Yaskawa INFORM job: DPRINT3D8.JBI

/JOB
//NAME DPRINT3D8
//POS
///NPOS 990,0,0,0,0,0
///TOOL 9
///POSTYPE PULSE
///PULSE
C00000=29490,52359,-120568,61658,-120234,-93746,0
C00001=29537,52361,-120565,61607,-120252,-93751,0
C00002=29592,52361,-120565,61546,-120272,-93759,0
C00003=29651,52358,-120574,61480,-120290,-93771,0
C00004=29730,52355,-120589,61392,-120313,-93786,0
C00005=29809,52348,-120612,61302,-120332,-93804,0
C00006=29942,52328,-120680,61146,-120353,-93842,0
C00007=30018,52314,-120729,61056,-120361,-93866,0
C00008=30112,52288,-120820,60939,-120358,-93905,0
C00009=30203,52259,-120919,60825,-120351,-93946,0
C00010=30285,52224,-121037,60719,-120333,-93990,0
C00011=30363,52187,-121164,60616,-120310,-94037,0
C00012=30429,52145,-121304,60523,-120276,-94086,0
C00013=30490,52102,-121452,60436,-120237,-94135,0
C00014=30538,52055,-121611,60361,-120190,-94186,0
C00015=30572,52018,-121739,60306,-120149,-94227,0
C00016=30580,52008,-121774,60292,-120138,-94237,0
C00017=30594,51982,-121860,60265,-120107,-94263,0
C00018=30605,51957,-121946,60241,-120076,-94288,0
C00019=30621,51904,-122127,60198,-120009,-94341,0
C00020=30624,51867,-122253,60178,-119957,-94376,0
C00021=30621,51830,-122380,60164,-119904,-94411,0
C00022=30618,51802,-122475,60155,-119864,-94437,0
C00023=30609,51776,-122563,60152,-119825,-94460,0
C00024=30600,51755,-122637,60152,-119791,-94479,0
C00025=30571,51703,-122814,60160,-119709,-94524,0
C00026=30542,51669,-122932,60176,-119650,-94553,0
C00027=30510,51638,-123039,60197,-119595,-94579,0
C00028=30482,51612,-123127,60216,-119549,-94600,0
C00029=30451,51588,-123208,60240,-119505,-94618,0
C00030=30396,51554,-123325,60285,-119439,-94643,0
C00031=30357,51531,-123404,60318,-119393,-94659,0
C00032=30314,51511,-123476,60355,-119349,-94673,0
C00033=30248,51483,-123570,60415,-119289,-94691,0
C00034=30201,51465,-123633,60459,-119247,-94702,0
C00035=30148,51448,-123692,60510,-119205,-94711,0
C00036=30074,51428,-123761,60583,-119152,-94720,0
C00037=30016,51413,-123811,60640,-119112,-94727,0
C00038=29954,51400,-123854,60703,-119074,-94730,0
C00039=29879,51388,-123894,60780,-119033,-94731,0
C00040=29815,51379,-123926,60847,-118999,-94732,0
C00041=29746,51372,-123949,60920,-118966,-94730,0
C00042=29673,51367,-123964,60998,-118936,-94724,0
C00043=29603,51364,-123975,61074,-118908,-94718,0
C00044=29535,51363,-123978,61148,-118885,-94709,0
C00045=29463,51364,-123971,61228,-118864,-94698,0
C00046=29411,51366,-123964,61286,-118849,-94689,0
C00047=29309,51372,-123940,61403,-118825,-94669,0
C00048=29207,51381,-123905,61519,-118804,-94646,0
C00049=29109,51397,-123850,61634,-118794,-94617,0
C00050=29015,51415,-123785,61747,-118788,-94586,0
C00051=28926,51438,-123701,61855,-118793,-94550,0
C00052=28842,51464,-123609,61960,-118801,-94513,0
C00053=28766,51495,-123499,62057,-118819,-94471,0
C00054=28695,51529,-123383,62150,-118841,-94429,0
C00055=28635,51566,-123252,62233,-118872,-94384,0
C00056=28581,51605,-123115,62311,-118908,-94338,0
C00057=28539,51647,-122969,62376,-118951,-94291,0
C00058=28503,51691,-122818,62435,-118997,-94243,0
C00059=28481,51736,-122661,62481,-119051,-94195,0
C00060=28464,51782,-122502,62520,-119109,-94148,0
C00061=28461,51829,-122341,62545,-119170,-94102,0
C00062=28463,51859,-122240,62556,-119210,-94073,0
C00063=28476,51924,-122018,62572,-119302,-94012,0
C00064=28493,51964,-121883,62572,-119360,-93976,0
C00065=28528,52017,-121701,62558,-119443,-93930,0
C00066=28561,52056,-121571,62539,-119506,-93897,0
C00067=28618,52106,-121405,62499,-119591,-93858,0
C00068=28668,52142,-121282,62461,-119657,-93830,0
C00069=28743,52185,-121137,62399,-119740,-93800,0
C00070=28808,52218,-121030,62342,-119805,-93779,0
C00071=28898,52253,-120912,62259,-119885,-93758,0
C00072=28977,52280,-120825,62185,-119948,-93744,0
C00073=29075,52306,-120741,62090,-120016,-93735,0
C00074=29171,52330,-120661,61995,-120081,-93726,0
C00075=25221,55476,-110646,67744,-122004,-90321,0
C00076=36362,52521,-120169,76431,-115202,-92037,0
C00077=36363,52459,-120191,76439,-115220,-92015,0
C00078=23322,59783,-98074,71828,-124780,-86450,0
C00079=23300,59778,-98087,71848,-124763,-86450,0
C00080=23207,59762,-98132,71934,-124696,-86448,0
C00081=23134,59755,-98149,72005,-124649,-86441,0
C00082=23037,59755,-98149,72103,-124591,-86425,0
C00083=22967,59761,-98132,72177,-124555,-86408,0
C00084=22871,59777,-98086,72281,-124511,-86380,0
C00085=22816,59791,-98047,72343,-124489,-86360,0
C00086=22729,59817,-97973,72444,-124458,-86325,0
C00087=22655,59848,-97887,72533,-124437,-86289,0
C00088=22584,59883,-97789,72621,-124421,-86250,0
C00089=22520,59926,-97670,72707,-124416,-86206,0
C00090=22458,59972,-97541,72791,-124413,-86159,0
C00091=22405,60025,-97394,72870,-124420,-86109,0
C00092=22356,60081,-97239,72947,-124432,-86057,0
C00093=22316,60142,-97070,73016,-124452,-86003,0
C00094=22280,60206,-96894,73082,-124478,-85948,0
C00095=22255,60273,-96709,73140,-124512,-85891,0
C00096=22235,60342,-96520,73194,-124549,-85835,0
C00097=22226,60412,-96326,73237,-124595,-85779,0
C00098=22221,60483,-96130,73276,-124643,-85722,0
C00099=22228,60555,-95934,73304,-124698,-85668,0
C00100=22235,60601,-95807,73320,-124736,-85633,0
C00101=22239,60626,-95740,73327,-124756,-85615,0
C00102=22260,60696,-95549,73341,-124818,-85565,0
C00103=22280,60753,-95392,73349,-124872,-85524,0
C00104=22317,60832,-95177,73351,-124950,-85469,0
C00105=22350,60886,-95029,73345,-125009,-85433,0
C00106=22403,60957,-94836,73326,-125091,-85387,0
C00107=22449,61008,-94699,73306,-125156,-85357,0
C00108=22516,61067,-94539,73269,-125238,-85322,0
C00109=22573,61109,-94424,73234,-125304,-85299,0
C00110=22650,61156,-94298,73180,-125384,-85277,0
C00111=22717,61189,-94210,73130,-125449,-85263,0
C00112=22802,61220,-94125,73061,-125523,-85253,0
C00113=22876,61242,-94068,72999,-125584,-85250,0
C00114=22965,61257,-94026,72917,-125651,-85253,0
C00115=22998,61262,-94015,72887,-125674,-85256,0
C00116=23044,61265,-94005,72844,-125705,-85261,0
C00117=23092,61265,-94006,72795,-125735,-85269,0
C00118=23153,61264,-94010,72735,-125772,-85281,0
C00119=23215,61259,-94025,72670,-125806,-85295,0
C00120=23304,61242,-94071,72574,-125849,-85324,0
C00121=23341,61233,-94096,72532,-125866,-85336,0
C00122=23382,61222,-94128,72485,-125882,-85353,0
C00123=23426,61205,-94174,72433,-125897,-85373,0
C00124=23485,61181,-94239,72362,-125916,-85401,0
C00125=23541,61155,-94311,72293,-125931,-85431,0
C00126=23615,61108,-94439,72195,-125943,-85480,0
C00127=23682,61057,-94580,72103,-125945,-85531,0
C00128=23740,60998,-94741,72014,-125938,-85586,0
C00129=23795,60936,-94911,71928,-125926,-85643,0
C00130=23805,60920,-94953,71910,-125920,-85657,0
C00131=23839,60868,-95097,71849,-125901,-85702,0
C00132=23879,60798,-95289,71773,-125874,-85763,0
C00133=23909,60724,-95491,71706,-125836,-85825,0
C00134=23933,60649,-95698,71644,-125795,-85887,0
C00135=23946,60571,-95910,71592,-125744,-85949,0
C00136=23947,60554,-95958,71582,-125731,-85962,0
C00137=23949,60494,-96123,71549,-125688,-86009,0
C00138=23946,60453,-96234,71532,-125656,-86040,0
C00139=23942,60416,-96335,71518,-125625,-86067,0
C00140=23926,60337,-96554,71493,-125556,-86125,0
C00141=23909,60283,-96701,71484,-125504,-86164,0
C00142=23887,60231,-96843,71480,-125452,-86200,0
C00143=23870,60192,-96951,71478,-125412,-86227,0
C00144=23849,60157,-97049,71481,-125373,-86251,0
C00145=23831,60129,-97125,71485,-125342,-86269,0
C00146=23781,60061,-97311,71501,-125260,-86313,0
C00147=23731,60007,-97459,71526,-125189,-86346,0
C00148=23666,59949,-97619,71563,-125107,-86380,0
C00149=23605,59906,-97737,71603,-125038,-86403,0
C00150=23529,59861,-97861,71657,-124959,-86425,0
C00151=23459,59829,-97949,71712,-124895,-86438,0
C00152=23402,59808,-98007,71760,-124844,-86445,0
C00153=23317,59765,-98126,71824,-124763,-86464,0
C00154=35332,54396,-113967,78226,-116318,-89994,0
C00155=36295,54803,-112729,77380,-117083,-89721,0
C00156=40947,51674,-122953,71228,-116241,-93341,0
C00157=33828,55772,-109747,58612,-126255,-91536,0
C00158=35387,54350,-114111,78152,-116309,-90043,0
C00159=35603,55084,-111856,78200,-116951,-89383,0
C00160=36476,55477,-110686,77450,-117670,-89127,0
C00161=42174,51641,-123098,69885,-116652,-93519,0
C00162=33600,55094,-111787,58512,-125351,-92026,0
C00163=34232,54514,-113579,79405,-115874,-89764,0
C00164=35133,54883,-112462,78609,-116575,-89515,0
C00165=34898,55093,-111816,78927,-116607,-89295,0
C00166=35366,55295,-111211,78521,-116983,-89162,0
C00167=35549,55132,-111710,78273,-116958,-89333,0
C00168=36108,54854,-112568,77592,-117031,-89652,0
C00169=34832,55352,-111030,57280,-126168,-92063,0
C00170=36949,53594,-116517,54010,-124665,-93861,0
C00171=39301,53631,-116452,73778,-117508,-91183,0
C00172=44249,56266,-108496,69707,-122168,-89514,0
C00173=34852,55334,-111085,79062,-116751,-89069,0
C00174=32937,57301,-105238,81692,-116962,-87111,0
C00175=36072,54385,-114015,77455,-116661,-90086,0
C00176=40136,51651,-123013,72093,-115916,-93273,0
C00177=48633,53267,-117848,63578,-120957,-92820,0
C00178=48723,53302,-117737,63496,-121033,-92802,0
C00179=48757,53314,-117700,63465,-121059,-92797,0
C00180=48805,53330,-117652,63419,-121097,-92790,0
C00181=48859,53343,-117610,63367,-121134,-92786,0
C00182=48926,53359,-117560,63301,-121178,-92782,0
C00183=48998,53374,-117515,63229,-121223,-92781,0
C00184=49105,53388,-117471,63119,-121282,-92785,0
C00185=49151,53393,-117456,63070,-121305,-92788,0
C00186=49204,53398,-117444,63015,-121330,-92792,0
C00187=49261,53399,-117440,62953,-121354,-92800,0
C00188=49339,53401,-117437,62868,-121386,-92810,0
C00189=49415,53400,-117441,62784,-121414,-92824,0
C00190=49524,53391,-117472,62661,-121444,-92848,0
C00191=49626,53378,-117520,62542,-121467,-92877,0
C00192=49724,53357,-117590,62425,-121478,-92911,0
C00193=49819,53332,-117670,62309,-121484,-92948,0
C00194=49839,53326,-117692,62283,-121484,-92958,0
C00195=49907,53302,-117771,62197,-121480,-92989,0
C00196=49992,53269,-117880,62088,-121470,-93032,0
C00197=50067,53230,-118008,61987,-121451,-93079,0
C00198=50138,53189,-118144,61889,-121426,-93128,0
C00199=50198,53143,-118293,61802,-121390,-93178,0
C00200=50209,53132,-118329,61784,-121381,-93190,0
C00201=50247,53094,-118453,61723,-121347,-93230,0
C00202=50268,53068,-118539,61688,-121322,-93257,0
C00203=50285,53043,-118620,61657,-121297,-93282,0
C00204=50316,52988,-118800,61597,-121238,-93336,0
C00205=50330,52950,-118927,61564,-121193,-93374,0
C00206=50337,52911,-119054,61536,-121147,-93410,0
C00207=50342,52881,-119151,61517,-121111,-93438,0
C00208=50342,52853,-119244,61504,-121074,-93464,0
C00209=50339,52830,-119318,61496,-121045,-93483,0
C00210=50326,52774,-119503,61483,-120967,-93533,0
C00211=50304,52726,-119660,61485,-120897,-93573,0
C00212=50269,52672,-119839,61498,-120814,-93617,0
C00213=50230,52628,-119982,61521,-120744,-93652,0
C00214=50175,52579,-120143,61558,-120660,-93688,0
C00215=50119,52540,-120271,61602,-120590,-93715,0
C00216=50043,52496,-120413,61664,-120507,-93744,0
C00217=49976,52465,-120515,61724,-120443,-93763,0
C00218=49884,52430,-120630,61809,-120364,-93782,0
C00219=49808,52406,-120707,61882,-120306,-93793,0
C00220=49702,52380,-120791,61986,-120236,-93801,0
C00221=49621,52365,-120839,62069,-120188,-93803,0
C00222=49505,52350,-120888,62189,-120127,-93800,0
C00223=49436,52344,-120906,62262,-120095,-93795,0
C00224=49322,52337,-120926,62384,-120047,-93785,0
C00225=49222,52336,-120924,62495,-120011,-93770,0
C00226=49121,52339,-120912,62607,-119980,-93753,0
C00227=49023,52349,-120879,62720,-119957,-93729,0
C00228=48926,52361,-120834,62832,-119939,-93703,0
C00229=48834,52380,-120769,62942,-119930,-93672,0
C00230=48744,52401,-120695,63050,-119926,-93638,0
C00231=48662,52428,-120602,63154,-119932,-93600,0
C00232=48584,52458,-120499,63253,-119942,-93560,0
C00233=48514,52493,-120382,63346,-119961,-93518,0
C00234=48450,52530,-120257,63433,-119984,-93473,0
C00235=48397,52571,-120118,63511,-120017,-93426,0
C00236=48349,52614,-119974,63583,-120053,-93379,0
C00237=48314,52660,-119821,63644,-120097,-93331,0
C00238=48294,52691,-119719,63680,-120128,-93299,0
C00239=48284,52708,-119665,63698,-120145,-93282,0
C00240=48265,52756,-119504,63741,-120198,-93234,0
C00241=48254,52798,-119367,63773,-120245,-93194,0
C00242=48249,52857,-119173,63806,-120315,-93138,0
C00243=48254,52900,-119033,63821,-120369,-93099,0
C00244=48272,52958,-118841,63828,-120448,-93048,0
C00245=48294,53002,-118699,63825,-120508,-93010,0
C00246=48334,53058,-118519,63807,-120591,-92965,0
C00247=48372,53100,-118383,63785,-120657,-92932,0
C00248=48432,53151,-118221,63743,-120739,-92895,0
C00249=48487,53190,-118095,63702,-120807,-92868,0
C00250=48559,53231,-117963,63642,-120884,-92842,0
C00251=48631,53272,-117834,63582,-120961,-92816,0
C00252=30446,52027,-121515,60488,-120235,-94120,0
C00253=30497,51984,-121663,60411,-120192,-94169,0
C00254=30538,51942,-121805,60346,-120149,-94214,0
C00255=30574,51891,-121979,60283,-120090,-94267,0
C00256=30585,51872,-122044,60262,-120068,-94286,0
C00257=30597,51845,-122135,60236,-120035,-94314,0
C00258=30605,51817,-122231,60215,-119998,-94341,0
C00259=30612,51782,-122353,60190,-119951,-94376,0
C00260=30615,51745,-122479,60170,-119899,-94412,0
C00261=30606,51692,-122661,60155,-119822,-94460,0
C00262=30599,51669,-122738,60152,-119788,-94481,0
C00263=30589,51644,-122824,60152,-119749,-94503,0
C00264=30572,51617,-122915,60158,-119706,-94527,0
C00265=30548,51581,-123038,60168,-119648,-94557,0
C00266=30520,51547,-123156,60184,-119589,-94586,0
C00267=30465,51501,-123316,60223,-119504,-94624,0
C00268=30402,51458,-123462,60273,-119424,-94655,0
C00269=30327,51420,-123592,60338,-119344,-94682,0
C00270=30246,51384,-123715,60411,-119267,-94705,0
C00271=30226,51377,-123740,60430,-119250,-94709,0
C00272=30156,51354,-123820,60497,-119194,-94722,0
C00273=30061,51326,-123916,60589,-119124,-94735,0
C00274=29958,51304,-123990,60692,-119058,-94743,0
C00275=29853,51285,-124056,60800,-118997,-94747,0
C00276=29742,51272,-124098,60916,-118943,-94744,0
C00277=29718,51270,-124104,60943,-118932,-94742,0
C00278=29630,51265,-124121,61037,-118896,-94736,0
C00279=29571,51263,-124125,61102,-118876,-94729,0
C00280=29517,51264,-124124,61162,-118858,-94722,0
C00281=29399,51267,-124111,61293,-118824,-94702,0
C00282=29319,51273,-124088,61385,-118807,-94685,0
C00283=29241,51281,-124057,61475,-118793,-94666,0
C00284=29181,51288,-124031,61544,-118784,-94651,0
C00285=29126,51297,-123998,61608,-118778,-94634,0
C00286=29084,51305,-123970,61659,-118776,-94621,0
C00287=28979,51329,-123886,61785,-118774,-94583,0
C00288=28894,51353,-123799,61889,-118780,-94547,0
C00289=28802,51385,-123685,62006,-118795,-94502,0
C00290=28732,51416,-123574,62097,-118815,-94462,0
C00291=28656,51457,-123434,62199,-118845,-94412,0
C00292=28603,51493,-123308,62273,-118877,-94369,0
C00293=28547,51540,-123145,62357,-118922,-94315,0
C00294=28512,51579,-123009,62413,-118963,-94272,0
C00295=28478,51630,-122831,62474,-119021,-94217,0
C00296=28461,51671,-122690,62511,-119071,-94174,0
C00297=28450,51726,-122502,62548,-119140,-94119,0
C00298=28451,51766,-122363,62565,-119195,-94080,0
C00299=28464,51822,-122174,62576,-119273,-94028,0
C00300=28482,51861,-122043,62575,-119331,-93993,0
C00301=28507,51907,-121886,62568,-119401,-93952,0
C00302=28519,51923,-121833,62562,-119425,-93939,0
C00303=28543,51952,-121735,62549,-119472,-93914,0
C00304=28585,51996,-121588,62523,-119544,-93878,0
C00305=28639,52037,-121450,62482,-119618,-93847,0
C00306=28698,52076,-121318,62436,-119690,-93818,0
C00307=28767,52112,-121199,62376,-119762,-93794,0
C00308=28815,52134,-121126,62334,-119808,-93780,0
C00309=28841,52145,-121088,62311,-119832,-93773,0
C00310=28923,52174,-120992,62234,-119898,-93758,0
C00311=29008,52200,-120906,62152,-119963,-93746,0
C00312=29100,52221,-120838,62062,-120022,-93739,0
C00313=29194,52239,-120780,61967,-120080,-93736,0
C00314=29292,52251,-120742,61865,-120130,-93740,0
C00315=29391,52260,-120713,61760,-120178,-93746,0
C00316=29491,52263,-120706,61651,-120217,-93758,0
C00317=29557,52263,-120707,61578,-120240,-93768,0
C00318=29591,52263,-120708,61540,-120252,-93773,0
C00319=29691,52257,-120729,61428,-120280,-93793,0
C00320=29774,52250,-120753,61334,-120300,-93812,0
C00321=29888,52236,-120805,61201,-120321,-93842,0
C00322=29968,52221,-120854,61106,-120330,-93868,0
C00323=30074,52196,-120941,60978,-120334,-93907,0
C00324=30150,52173,-121018,60883,-120330,-93940,0
C00325=30242,52139,-121134,60766,-120317,-93985,0
C00326=30309,52110,-121236,60678,-120299,-94023,0
C00327=30385,52068,-121377,60574,-120268,-94073,0
C00328=30386,52067,-121378,60573,-120268,-94074,0
C00329=30509,52006,-121589,60409,-120227,-94150,0
C00330=25260,55430,-110634,67719,-122054,-90298,0
C00331=36363,52459,-120191,76439,-115220,-92015,0
C00332=39710,59332,-99593,75775,-122140,-86293,0
C00333=39635,59289,-99712,75830,-122067,-86316,0
C00334=39558,59250,-99820,75890,-121994,-86337,0
C00335=39474,59220,-99903,75960,-121925,-86348,0
C00336=39455,59215,-99917,75977,-121910,-86350,0
C00337=39387,59197,-99964,76037,-121860,-86354,0
C00338=39341,59189,-99986,76079,-121827,-86354,0
C00339=39298,59184,-100001,76120,-121798,-86352,0
C00340=39204,59176,-100021,76211,-121738,-86344,0
C00341=39138,59176,-100019,76276,-121700,-86334,0
C00342=39074,59180,-100006,76342,-121665,-86322,0
C00343=39024,59184,-99994,76393,-121638,-86311,0
C00344=38978,59192,-99972,76442,-121616,-86299,0
C00345=38942,59199,-99951,76481,-121600,-86288,0
C00346=38852,59222,-99886,76581,-121562,-86257,0
C00347=38777,59249,-99809,76667,-121536,-86224,0
C00348=38694,59286,-99704,76765,-121512,-86182,0
C00349=38629,59323,-99597,76846,-121498,-86142,0
C00350=38556,59374,-99455,76940,-121489,-86091,0
C00351=38503,59420,-99325,77012,-121488,-86046,0
C00352=38445,59482,-99150,77098,-121492,-85988,0
C00353=38405,59535,-99002,77159,-121504,-85940,0
C00354=38362,59606,-98804,77232,-121523,-85877,0
C00355=38337,59663,-98644,77282,-121545,-85827,0
C00356=38312,59742,-98426,77340,-121581,-85761,0
C00357=38301,59800,-98263,77377,-121611,-85712,0
C00358=38295,59882,-98036,77418,-121660,-85646,0
C00359=38298,59940,-97876,77440,-121698,-85600,0
C00360=38305,60010,-97683,77463,-121746,-85546,0
C00361=38310,60033,-97618,77469,-121765,-85527,0
C00362=38321,60078,-97493,77478,-121799,-85493,0
C00363=38342,60146,-97306,77486,-121855,-85442,0
C00364=38373,60212,-97127,77484,-121915,-85395,0
C00365=38410,60275,-96952,77476,-121977,-85350,0
C00366=38455,60334,-96790,77458,-122043,-85309,0
C00367=38487,60372,-96688,77443,-122085,-85285,0
C00368=38505,60391,-96635,77434,-122108,-85271,0
C00369=38562,60442,-96496,77400,-122176,-85240,0
C00370=38623,60489,-96367,77361,-122243,-85211,0
C00371=38691,60530,-96257,77313,-122310,-85190,0
C00372=38761,60567,-96158,77261,-122376,-85171,0
C00373=38836,60595,-96081,77200,-122440,-85159,0
C00374=38912,60619,-96016,77136,-122503,-85152,0
C00375=38992,60634,-95976,77065,-122562,-85152,0
C00376=39044,60642,-95957,77017,-122599,-85154,0
C00377=39072,60645,-95948,76991,-122618,-85155,0
C00378=39153,60648,-95941,76914,-122670,-85165,0
C00379=39221,60648,-95943,76847,-122713,-85175,0
C00380=39316,60639,-95969,76750,-122765,-85196,0
C00381=39384,60627,-96003,76678,-122799,-85216,0
C00382=39475,60602,-96073,76578,-122839,-85249,0
C00383=39542,60578,-96141,76501,-122865,-85278,0
C00384=39624,60539,-96250,76403,-122890,-85322,0
C00385=39686,60503,-96350,76326,-122904,-85360,0
C00386=39758,60450,-96496,76231,-122914,-85412,0
C00387=39814,60401,-96632,76153,-122916,-85459,0
C00388=39869,60340,-96801,76071,-122910,-85516,0
C00389=39913,60284,-96956,76002,-122900,-85566,0
C00390=39956,60213,-97153,75927,-122878,-85629,0
C00391=39970,60187,-97225,75902,-122870,-85651,0
C00392=39987,60149,-97330,75868,-122855,-85684,0
C00393=40001,60109,-97443,75836,-122836,-85718,0
C00394=40016,60058,-97584,75797,-122811,-85761,0
C00395=40029,60004,-97732,75760,-122783,-85805,0
C00396=40036,59925,-97950,75717,-122734,-85869,0
C00397=40037,59892,-98043,75701,-122713,-85896,0
C00398=40036,59854,-98148,75685,-122686,-85925,0
C00399=40031,59813,-98261,75672,-122655,-85957,0
C00400=40022,59758,-98414,75656,-122613,-86000,0
C00401=40009,59705,-98561,75645,-122569,-86040,0
C00402=39979,59631,-98767,75641,-122501,-86095,0
C00403=39941,59562,-98957,75647,-122432,-86143,0
C00404=39893,59499,-99133,75667,-122360,-86187,0
C00405=39839,59438,-99302,75693,-122287,-86228,0
C00406=39773,59380,-99460,75734,-122209,-86264,0
C00407=39713,59315,-99642,75764,-122130,-86307,0
C00408=39713,59261,-99663,75774,-122146,-86289,0
C00409=23871,60661,-95543,71751,-125822,-85809,0
C00410=23879,60642,-95595,71733,-125813,-85825,0
C00411=23895,60596,-95721,71693,-125789,-85863,0
C00412=23905,60552,-95840,71661,-125762,-85898,0
C00413=23918,60488,-96016,71616,-125722,-85950,0
C00414=23923,60446,-96131,71590,-125693,-85983,0
C00415=23923,60403,-96250,71567,-125660,-86016,0
C00416=23923,60350,-96395,71541,-125620,-86056,0
C00417=23917,60294,-96548,71519,-125575,-86099,0
C00418=23899,60215,-96764,71497,-125505,-86156,0
C00419=23890,60182,-96857,71490,-125474,-86181,0
C00420=23877,60145,-96958,71485,-125437,-86207,0
C00421=23859,60107,-97062,71484,-125398,-86233,0
C00422=23833,60056,-97203,71484,-125344,-86268,0
C00423=23803,60006,-97338,71490,-125289,-86301,0
C00424=23738,59925,-97562,71515,-125189,-86352,0
C00425=23696,59880,-97685,71536,-125130,-86380,0
C00426=23629,59829,-97826,71578,-125052,-86408,0
C00427=23558,59782,-97956,71626,-124974,-86433,0
C00428=23481,59743,-98063,71685,-124899,-86450,0
C00429=23401,59708,-98158,71749,-124826,-86463,0
C00430=23316,59683,-98226,71823,-124758,-86468,0
C00431=23229,59663,-98282,71901,-124691,-86470,0
C00432=23140,59652,-98309,71986,-124632,-86463,0
C00433=23070,59648,-98321,72054,-124588,-86455,0
C00434=23050,59647,-98324,72074,-124575,-86452,0
C00435=23005,59649,-98316,72121,-124551,-86442,0
C00436=22961,59654,-98302,72168,-124528,-86431,0
C00437=22873,59667,-98265,72263,-124487,-86406,0
C00438=22826,59678,-98234,72315,-124467,-86390,0
C00439=22788,59689,-98203,72359,-124454,-86375,0
C00440=22701,59718,-98122,72460,-124425,-86338,0
C00441=22644,59744,-98050,72530,-124410,-86309,0
C00442=22591,59772,-97971,72598,-124400,-86278,0
C00443=22550,59795,-97906,72650,-124393,-86253,0
C00444=22513,59820,-97837,72699,-124390,-86227,0
C00445=22488,59840,-97782,72734,-124389,-86208,0
C00446=22421,59896,-97627,72828,-124391,-86153,0
C00447=22372,59949,-97479,72903,-124401,-86103,0
C00448=22320,60016,-97295,72987,-124419,-86043,0
C00449=22285,60075,-97130,73052,-124441,-85991,0
C00450=22249,60150,-96923,73123,-124474,-85926,0
C00451=22229,60213,-96749,73174,-124508,-85874,0
C00452=22212,60294,-96528,73230,-124556,-85809,0
C00453=22206,60358,-96352,73267,-124598,-85758,0
C00454=22207,60441,-96123,73306,-124658,-85694,0
C00455=22216,60503,-95953,73328,-124708,-85647,0
C00456=22236,60586,-95727,73349,-124779,-85587,0
C00457=22257,60644,-95568,73356,-124833,-85546,0
C00458=22301,60733,-95326,73355,-124924,-85485,0
C00459=22325,60776,-95210,73352,-124968,-85456,0
C00460=22366,60838,-95040,73342,-125037,-85415,0
C00461=22416,60896,-94884,73320,-125109,-85379,0
C00462=22470,60950,-94736,73294,-125181,-85346,0
C00463=22531,60998,-94607,73257,-125252,-85320,0
C00464=22595,61042,-94486,73215,-125322,-85297,0
C00465=22665,61079,-94388,73164,-125391,-85281,0
C00466=22737,61111,-94301,73109,-125459,-85268,0
C00467=22763,61120,-94278,73087,-125481,-85266,0
C00468=22813,61135,-94237,73045,-125523,-85263,0
C00469=22890,61154,-94186,72978,-125584,-85262,0
C00470=22970,61164,-94161,72904,-125641,-85268,0
C00471=23050,61169,-94147,72827,-125693,-85278,0
C00472=23130,61165,-94160,72745,-125739,-85295,0
C00473=23209,61156,-94185,72662,-125782,-85315,0
C00474=23287,61138,-94236,72575,-125816,-85343,0
C00475=23363,61115,-94299,72488,-125847,-85373,0
C00476=23400,61101,-94337,72444,-125860,-85391,0
C00477=23449,61082,-94388,72386,-125876,-85414,0
C00478=23498,61059,-94452,72325,-125890,-85440,0
C00479=23543,61033,-94524,72267,-125898,-85467,0
C00480=23590,61003,-94604,72205,-125906,-85498,0
C00481=23632,60973,-94688,72148,-125908,-85529,0
C00482=23670,60940,-94778,72094,-125907,-85560,0
C00483=23713,60900,-94887,72030,-125904,-85599,0
C00484=23746,60864,-94985,71979,-125898,-85632,0
C00485=23775,60826,-95090,71930,-125888,-85666,0
C00486=23811,60777,-95225,71870,-125873,-85710,0
C00487=23839,60729,-95356,71817,-125854,-85751,0
C00488=23893,60658,-95551,71726,-125834,-85816,0
C00489=35332,54337,-113989,78234,-116334,-89973,0
C00490=36295,54745,-112751,77388,-117100,-89701,0
C00491=40947,51611,-122976,71236,-116264,-93318,0
C00492=33829,55715,-109769,58624,-126282,-91519,0
C00493=35387,54291,-114133,78160,-116326,-90023,0
C00494=35603,55027,-111878,78208,-116967,-89362,0
C00495=36476,55419,-110708,77458,-117686,-89107,0
C00496=42175,51578,-123121,69893,-116676,-93497,0
C00497=33600,55037,-111809,58523,-125379,-92008,0
C00498=34232,54455,-113601,79413,-115890,-89743,0
C00499=35133,54825,-112483,78617,-116591,-89495,0
C00500=34898,55035,-111838,78935,-116623,-89275,0
C00501=35367,55238,-111233,78529,-116999,-89142,0
C00502=35549,55074,-111732,78281,-116975,-89312,0
C00503=36109,54796,-112590,77600,-117048,-89632,0
C00504=34832,55294,-111052,57291,-126196,-92045,0
C00505=36934,53545,-116504,54043,-124705,-93831,0
C00506=39301,53571,-116475,73786,-117528,-91162,0
C00507=44220,56190,-108573,69740,-122156,-89507,0
C00508=34852,55276,-111107,79070,-116766,-89049,0
C00509=32950,57232,-105299,81683,-116975,-87105,0
C00510=36072,54326,-114037,77463,-116677,-90066,0
C00511=40137,51587,-123035,72101,-115939,-93251,0
C00512=48524,53119,-118152,63666,-120835,-92863,0
C00513=48595,53155,-118037,63606,-120905,-92842,0
C00514=48669,53189,-117930,63540,-120974,-92822,0
C00515=48752,53217,-117840,63463,-121039,-92810,0
C00516=48837,53243,-117760,63382,-121104,-92799,0
C00517=48928,53263,-117698,63292,-121161,-92796,0
C00518=49021,53279,-117647,63198,-121218,-92795,0
C00519=49116,53290,-117616,63098,-121266,-92801,0
C00520=49213,53297,-117597,62996,-121312,-92810,0
C00521=49262,53299,-117592,62943,-121332,-92816,0
C00522=49326,53301,-117587,62874,-121359,-92825,0
C00523=49393,53300,-117592,62800,-121383,-92836,0
C00524=49458,53296,-117607,62727,-121403,-92850,0
C00525=49526,53290,-117625,62649,-121423,-92865,0
C00526=49590,53283,-117652,62576,-121438,-92883,0
C00527=49650,53272,-117686,62505,-121447,-92901,0
C00528=49720,53259,-117731,62422,-121458,-92924,0
C00529=49777,53246,-117776,62353,-121463,-92945,0
C00530=49831,53230,-117829,62285,-121463,-92969,0
C00531=49899,53209,-117899,62201,-121463,-92998,0
C00532=49953,53188,-117967,62132,-121458,-93025,0
C00533=50006,53164,-118047,62062,-121447,-93056,0
C00534=50052,53142,-118119,62001,-121437,-93082,0
C00535=50097,53117,-118201,61939,-121423,-93112,0
C00536=50134,53092,-118281,61887,-121406,-93140,0
C00537=50186,53055,-118403,61812,-121378,-93182,0
C00538=50216,53030,-118487,61766,-121358,-93209,0
C00539=50242,53002,-118577,61724,-121332,-93238,0
C00540=50273,52968,-118688,61674,-121301,-93273,0
C00541=50301,52931,-118809,61626,-121265,-93311,0
C00542=50329,52876,-118989,61569,-121205,-93365,0
C00543=50339,52852,-119069,61546,-121178,-93389,0
C00544=50347,52825,-119157,61524,-121146,-93414,0
C00545=50350,52796,-119252,61507,-121111,-93441,0
C00546=50354,52757,-119381,61484,-121061,-93477,0
C00547=50352,52717,-119511,61468,-121010,-93513,0
C00548=50331,52648,-119739,61458,-120913,-93573,0
C00549=50312,52608,-119870,61459,-120856,-93606,0
C00550=50271,52558,-120035,61481,-120775,-93646,0
C00551=50224,52508,-120196,61510,-120695,-93684,0
C00552=50164,52463,-120344,61555,-120614,-93717,0
C00553=50097,52420,-120487,61607,-120534,-93747,0
C00554=50020,52381,-120613,61675,-120457,-93771,0
C00555=49938,52345,-120730,61748,-120381,-93791,0
C00556=49846,52315,-120829,61835,-120310,-93806,0
C00557=49773,52293,-120899,61906,-120256,-93815,0
C00558=49751,52287,-120919,61927,-120241,-93818,0
C00559=49700,52277,-120952,61979,-120209,-93819,0
C00560=49648,52268,-120980,62032,-120179,-93820,0
C00561=49543,52253,-121028,62141,-120122,-93819,0
C00562=49485,52247,-121045,62202,-120095,-93815,0
C00563=49435,52244,-121055,62255,-120073,-93811,0
C00564=49321,52239,-121068,62378,-120027,-93798,0
C00565=49242,52240,-121064,62466,-120001,-93786,0
C00566=49166,52243,-121050,62552,-119979,-93771,0
C00567=49105,52247,-121036,62620,-119961,-93759,0
C00568=49049,52252,-121015,62684,-119950,-93746,0
C00569=49008,52258,-120997,62732,-119942,-93735,0
C00570=48900,52275,-120936,62859,-119926,-93702,0
C00571=48812,52295,-120867,62965,-119920,-93670,0
C00572=48713,52322,-120773,63087,-119920,-93630,0
C00573=48637,52349,-120680,63183,-119928,-93592,0
C00574=48551,52387,-120553,63295,-119944,-93545,0
C00575=48490,52420,-120441,63377,-119965,-93504,0
C00576=48421,52465,-120289,63473,-119997,-93452,0
C00577=48376,52503,-120160,63541,-120028,-93409,0
C00578=48327,52555,-119987,63618,-120075,-93353,0
C00579=48299,52596,-119852,63668,-120115,-93311,0
C00580=48272,52653,-119664,63724,-120175,-93254,0
C00581=48262,52695,-119527,63755,-120224,-93213,0
C00582=48258,52745,-119362,63783,-120283,-93166,0
C00583=48261,52795,-119197,63803,-120345,-93120,0
C00584=48270,52845,-119033,63816,-120410,-93075,0
C00585=48292,52895,-118872,63815,-120479,-93032,0
C00586=48320,52944,-118714,63807,-120548,-92992,0
C00587=48360,52990,-118563,63785,-120619,-92955,0
C00588=48406,53036,-118416,63757,-120691,-92920,0
C00589=48461,53077,-118285,63716,-120761,-92891,0
C00590=48514,53135,-118098,63685,-120851,-92847,0
C00591=30390,51969,-121522,60562,-120250,-94088,0
C00592=30409,51955,-121571,60534,-120236,-94105,0
C00593=30454,51912,-121717,60465,-120194,-94151,0
C00594=30492,51868,-121867,60402,-120147,-94198,0
C00595=30518,51822,-122023,60351,-120091,-94245,0
C00596=30538,51775,-122182,60308,-120034,-94292,0
C00597=30544,51728,-122343,60279,-119970,-94337,0
C00598=30544,51681,-122505,60257,-119904,-94383,0
C00599=30530,51634,-122663,60251,-119834,-94424,0
C00600=30518,51605,-122761,60251,-119790,-94450,0
C00601=30483,51542,-122978,60261,-119689,-94505,0
C00602=30452,51505,-123106,60277,-119626,-94536,0
C00603=30398,51456,-123273,60314,-119539,-94576,0
C00604=30350,51421,-123394,60351,-119473,-94603,0
C00605=30276,51378,-123540,60413,-119388,-94633,0
C00606=30212,51347,-123646,60470,-119324,-94654,0
C00607=30121,51312,-123766,60555,-119243,-94676,0
C00608=30043,51287,-123853,60630,-119182,-94689,0
C00609=29938,51261,-123941,60734,-119111,-94700,0
C00610=29847,51242,-124003,60825,-119055,-94705,0
C00611=29734,51226,-124058,60943,-118995,-94705,0
C00612=29635,51216,-124092,61048,-118948,-94701,0
C00613=29517,51210,-124110,61176,-118902,-94691,0
C00614=29473,51209,-124113,61224,-118886,-94686,0
C00615=29413,51208,-124113,61290,-118866,-94678,0
C00616=29351,51211,-124104,61360,-118849,-94667,0
C00617=29272,51215,-124089,61449,-118828,-94653,0
C00618=29191,51221,-124066,61540,-118811,-94635,0
C00619=29079,51236,-124012,61671,-118795,-94606,0
C00620=29030,51243,-123985,61728,-118789,-94591,0
C00621=28975,51253,-123948,61794,-118786,-94573,0
C00622=28876,51277,-123864,61913,-118786,-94536,0
C00623=28828,51290,-123818,61972,-118788,-94517,0
C00624=28782,51304,-123769,62030,-118792,-94496,0
C00625=28763,51312,-123742,62054,-118796,-94487,0
C00626=28699,51338,-123649,62136,-118811,-94452,0
C00627=28622,51374,-123522,62237,-118835,-94405,0
C00628=28557,51415,-123379,62328,-118870,-94356,0
C00629=28498,51458,-123231,62412,-118908,-94306,0
C00630=28452,51504,-123070,62483,-118955,-94254,0
C00631=28413,51552,-122907,62548,-119005,-94202,0
C00632=28388,51601,-122734,62597,-119064,-94151,0
C00633=28371,51652,-122562,62640,-119126,-94099,0
C00634=28371,51691,-122430,62657,-119178,-94061,0
C00635=28382,51757,-122204,62675,-119269,-93999,0
C00636=28398,51794,-122079,62674,-119323,-93966,0
C00637=28420,51830,-121956,62667,-119379,-93934,0
C00638=28437,51857,-121864,62660,-119420,-93910,0
C00639=28458,51882,-121782,62649,-119459,-93889,0
C00640=28478,51902,-121714,62636,-119494,-93873,0
C00641=28532,51951,-121551,62599,-119577,-93834,0
C00642=28576,51982,-121445,62565,-119633,-93811,0
C00643=28622,52010,-121351,62528,-119687,-93790,0
C00644=28661,52034,-121274,62496,-119731,-93774,0
C00645=28702,52054,-121205,62459,-119772,-93760,0
C00646=28771,52084,-121107,62397,-119835,-93743,0
C00647=28819,52103,-121043,62354,-119878,-93731,0
C00648=28870,52120,-120987,62305,-119918,-93722,0
C00649=28945,52142,-120916,62233,-119972,-93714,0
C00650=29001,52157,-120868,62178,-120012,-93707,0
C00651=29059,52169,-120828,62121,-120049,-93704,0
C00652=29136,52182,-120784,62042,-120094,-93703,0
C00653=29198,52192,-120754,61979,-120128,-93704,0
C00654=29262,52199,-120731,61911,-120160,-93706,0
C00655=29338,52204,-120715,61831,-120194,-93712,0
C00656=29404,52208,-120704,61760,-120222,-93719,0
C00657=29470,52209,-120702,61687,-120248,-93728,0
C00658=29542,52207,-120710,61608,-120271,-93740,0
C00659=29609,52204,-120720,61533,-120291,-93753,0
C00660=29677,52199,-120739,61455,-120307,-93768,0
C00661=29741,52191,-120767,61381,-120320,-93785,0
C00662=29822,52179,-120807,61286,-120333,-93808,0
C00663=29945,52157,-120885,61141,-120346,-93847,0
C00664=29977,52150,-120908,61102,-120349,-93858,0
C00665=30063,52125,-120991,60996,-120346,-93894,0
C00666=30146,52099,-121083,60891,-120341,-93931,0
C00667=30222,52067,-121191,60793,-120323,-93972,0
C00668=30293,52033,-121306,60699,-120303,-94014,0
C00669=30330,52009,-121385,60647,-120283,-94042,0
C00670=30426,51970,-121519,60523,-120264,-94093,0
C00671=25298,55384,-110622,67694,-122106,-90276,0
C00672=36363,52397,-120214,76446,-115238,-91993,0
C00673=38424,59383,-99298,77108,-121466,-86003,0
C00674=38411,59397,-99261,77127,-121467,-85990,0
C00675=38361,59458,-99088,77203,-121477,-85933,0
C00676=38315,59523,-98908,77276,-121491,-85875,0
C00677=38281,59592,-98714,77339,-121515,-85815,0
C00678=38252,59663,-98516,77398,-121543,-85754,0
C00679=38241,59719,-98361,77433,-121571,-85708,0
C00680=38231,59816,-98092,77485,-121627,-85629,0
C00681=38233,59871,-97941,77507,-121663,-85585,0
C00682=38240,59926,-97790,77524,-121701,-85543,0
C00683=38245,59967,-97676,77536,-121731,-85510,0
C00684=38255,60005,-97572,77543,-121761,-85482,0
C00685=38265,60036,-97484,77547,-121786,-85458,0
C00686=38294,60112,-97275,77551,-121852,-85402,0
C00687=38321,60163,-97137,77547,-121900,-85366,0
C00688=38350,60209,-97010,77539,-121946,-85333,0
C00689=38374,60247,-96907,77531,-121985,-85307,0
C00690=38402,60281,-96812,77519,-122023,-85284,0
C00691=38449,60331,-96675,77495,-122084,-85251,0
C00692=38482,60365,-96584,77478,-122125,-85230,0
C00693=38518,60395,-96501,77456,-122167,-85210,0
C00694=38572,60434,-96394,77420,-122224,-85188,0
C00695=38613,60462,-96319,77393,-122267,-85172,0
C00696=38655,60486,-96253,77362,-122308,-85159,0
C00697=38714,60514,-96177,77317,-122362,-85145,0
C00698=38760,60535,-96121,77281,-122403,-85136,0
C00699=38809,60553,-96074,77241,-122445,-85129,0
C00700=38869,60569,-96031,77190,-122492,-85126,0
C00701=38920,60582,-95997,77145,-122532,-85123,0
C00702=38973,60591,-95973,77097,-122570,-85124,0
C00703=39031,60596,-95960,77044,-122609,-85129,0
C00704=39085,60600,-95950,76992,-122645,-85133,0
C00705=39141,60599,-95953,76937,-122679,-85142,0
C00706=39194,60595,-95966,76883,-122709,-85154,0
C00707=39235,60591,-95977,76842,-122732,-85163,0
C00708=39315,60579,-96012,76758,-122773,-85184,0
C00709=39393,60562,-96060,76674,-122811,-85209,0
C00710=39469,60536,-96131,76588,-122841,-85241,0
C00711=39542,60507,-96214,76503,-122868,-85275,0
C00712=39611,60469,-96320,76418,-122885,-85315,0
C00713=39677,60427,-96435,76335,-122899,-85358,0
C00714=39735,60378,-96570,76255,-122903,-85405,0
C00715=39790,60327,-96714,76177,-122902,-85455,0
C00716=39837,60269,-96873,76104,-122894,-85507,0
C00717=39880,60209,-97039,76035,-122880,-85561,0
C00718=39913,60145,-97217,75973,-122857,-85617,0
C00719=39942,60079,-97399,75915,-122831,-85673,0
C00720=39960,60011,-97588,75866,-122796,-85729,0
C00721=39973,59942,-97779,75822,-122759,-85786,0
C00722=39975,59872,-97971,75788,-122713,-85842,0
C00723=39974,59829,-98090,75770,-122684,-85875,0
C00724=39963,59733,-98357,75737,-122613,-85950,0
C00725=39949,59675,-98516,75725,-122565,-85994,0
C00726=39921,59597,-98732,75718,-122495,-86051,0
C00727=39893,59541,-98887,75720,-122441,-86092,0
C00728=39847,59471,-99082,75735,-122367,-86141,0
C00729=39805,59419,-99225,75753,-122307,-86176,0
C00730=39743,59358,-99395,75788,-122229,-86216,0
C00731=39688,59313,-99519,75822,-122166,-86244,0
C00732=39613,59264,-99655,75875,-122089,-86272,0
C00733=39547,59227,-99755,75925,-122025,-86291,0
C00734=39462,59192,-99853,75994,-121951,-86308,0
C00735=39387,59166,-99923,76058,-121890,-86317,0
C00736=39295,59145,-99980,76140,-121822,-86320,0
C00737=39260,59139,-99998,76171,-121798,-86321,0
C00738=39213,59132,-100015,76215,-121766,-86319,0
C00739=39163,59129,-100023,76264,-121733,-86315,0
C00740=39099,59126,-100030,76326,-121694,-86308,0
C00741=39034,59126,-100027,76392,-121657,-86298,0
C00742=38940,59136,-99999,76489,-121608,-86276,0
C00743=38899,59142,-99981,76533,-121588,-86266,0
C00744=38852,59151,-99955,76583,-121566,-86251,0
C00745=38766,59175,-99887,76679,-121531,-86220,0
C00746=38724,59188,-99848,76726,-121516,-86203,0
C00747=38683,59204,-99804,76774,-121503,-86185,0
C00748=38607,59244,-99689,76867,-121484,-86141,0
C00749=38535,59289,-99564,76958,-121470,-86095,0
C00750=38482,59332,-99443,77028,-121467,-86053,0
C00751=38404,59380,-99308,77127,-121452,-86003,0
C00752=38404,59326,-99329,77136,-121467,-85984,0
C00753=23799,60690,-95341,71876,-125857,-85717,0
C00754=23811,60667,-95404,71851,-125847,-85737,0
C00755=23838,60599,-95590,71790,-125813,-85793,0
C00756=23860,60529,-95779,71733,-125775,-85850,0
C00757=23872,60458,-95974,71685,-125729,-85907,0
C00758=23879,60387,-96170,71643,-125679,-85962,0
C00759=23874,60316,-96365,71611,-125623,-86016,0
C00760=23865,60245,-96560,71585,-125564,-86069,0
C00761=23858,60221,-96625,71580,-125542,-86087,0
C00762=23845,60176,-96749,71571,-125500,-86119,0
C00763=23820,60108,-96934,71562,-125434,-86166,0
C00764=23781,60035,-97135,71564,-125356,-86216,0
C00765=23755,59991,-97255,71569,-125307,-86245,0
C00766=23725,59951,-97366,71579,-125259,-86271,0
C00767=23693,59911,-97477,71591,-125210,-86297,0
C00768=23658,59873,-97579,71608,-125160,-86320,0
C00769=23621,59840,-97670,71630,-125113,-86339,0
C00770=23577,59804,-97771,71656,-125059,-86360,0
C00771=23536,59774,-97851,71683,-125013,-86376,0
C00772=23491,59748,-97922,71715,-124967,-86388,0
C00773=23437,59719,-98004,71755,-124913,-86402,0
C00774=23391,59697,-98062,71792,-124870,-86410,0
C00775=23342,59680,-98110,71832,-124828,-86416,0
C00776=23278,59659,-98168,71886,-124775,-86421,0
C00777=23229,59646,-98202,71930,-124736,-86423,0
C00778=23179,59637,-98226,71976,-124701,-86421,0
C00779=23107,59627,-98254,72044,-124650,-86417,0
C00780=23058,59623,-98264,72092,-124619,-86412,0
C00781=23007,59623,-98263,72143,-124589,-86404,0
C00782=22930,59625,-98257,72221,-124545,-86390,0
C00783=22883,59629,-98245,72271,-124521,-86378,0
C00784=22834,59638,-98221,72325,-124500,-86363,0
C00785=22773,59649,-98188,72391,-124472,-86344,0
C00786=22712,59665,-98144,72461,-124448,-86322,0
C00787=22626,59696,-98056,72562,-124420,-86283,0
C00788=22591,59711,-98015,72605,-124411,-86266,0
C00789=22552,59730,-97963,72653,-124402,-86245,0
C00790=22512,59753,-97898,72705,-124396,-86220,0
C00791=22459,59786,-97806,72774,-124388,-86186,0
C00792=22410,59821,-97709,72840,-124385,-86150,0
C00793=22346,59878,-97550,72932,-124389,-86095,0
C00794=22292,59939,-97381,73015,-124402,-86039,0
C00795=22249,60006,-97196,73091,-124425,-85980,0
C00796=22211,60076,-97005,73163,-124452,-85920,0
C00797=22204,60093,-96958,73178,-124460,-85905,0
C00798=22183,60149,-96802,73225,-124488,-85858,0
C00799=22161,60224,-96597,73283,-124529,-85796,0
C00800=22151,60301,-96384,73331,-124579,-85735,0
C00801=22147,60379,-96171,73373,-124632,-85674,0
C00802=22154,60457,-95958,73403,-124691,-85615,0
C00803=22159,60482,-95890,73411,-124711,-85597,0
C00804=22170,60534,-95747,73425,-124756,-85559,0
C00805=22183,60573,-95641,73431,-124791,-85531,0
C00806=22197,60608,-95544,73434,-124825,-85505,0
C00807=22232,60684,-95338,73437,-124899,-85453,0
C00808=22263,60734,-95202,73430,-124953,-85420,0
C00809=22297,60782,-95072,73420,-125009,-85389,0
C00810=22324,60818,-94974,73411,-125050,-85365,0
C00811=22352,60850,-94888,73399,-125090,-85346,0
C00812=22376,60874,-94823,73387,-125122,-85332,0
C00813=22440,60933,-94663,73352,-125203,-85297,0
C00814=22489,60969,-94565,73321,-125259,-85278,0
C00815=22538,61000,-94482,73288,-125311,-85263,0
C00816=22578,61025,-94415,73260,-125353,-85250,0
C00817=22621,61046,-94357,73229,-125395,-85241,0
C00818=22647,61057,-94326,73208,-125419,-85237,0
C00819=22732,61090,-94238,73140,-125495,-85226,0
C00820=22804,61110,-94186,73078,-125553,-85224,0
C00821=22895,61127,-94141,72998,-125621,-85226,0
C00822=22968,61133,-94124,72928,-125671,-85234,0
C00823=23061,61134,-94124,72836,-125729,-85249,0
C00824=23132,61128,-94142,72762,-125768,-85267,0
C00825=23224,61111,-94187,72663,-125813,-85295,0
C00826=23289,61093,-94237,72588,-125841,-85320,0
C00827=23378,61060,-94327,72484,-125872,-85360,0
C00828=23426,61037,-94390,72423,-125884,-85387,0
C00829=23505,60995,-94506,72324,-125901,-85433,0
C00830=23569,60951,-94626,72238,-125910,-85477,0
C00831=23609,60921,-94710,72182,-125912,-85508,0
C00832=23630,60904,-94755,72153,-125912,-85524,0
C00833=23684,60850,-94903,72072,-125905,-85574,0
C00834=23734,60793,-95058,71993,-125893,-85626,0
C00835=23759,60755,-95163,71948,-125881,-85660,0
C00836=23827,60688,-95345,71846,-125873,-85723,0
C00837=35333,54278,-114010,78241,-116351,-89952,0
C00838=36295,54687,-112773,77397,-117117,-89680,0
C00839=40947,51547,-122999,71244,-116286,-93296,0
C00840=33829,55658,-109791,58635,-126308,-91502,0
C00841=35387,54232,-114155,78168,-116343,-90002,0
C00842=35603,54969,-111900,78216,-116983,-89341,0
C00843=36476,55362,-110730,77467,-117702,-89087,0
C00844=42175,51514,-123142,69902,-116700,-93476,0
C00845=33601,54979,-111831,58534,-125406,-91991,0
C00846=34232,54397,-113623,79420,-115906,-89721,0
C00847=35134,54767,-112505,78625,-116607,-89474,0
C00848=34899,54978,-111859,78943,-116638,-89254,0
C00849=35367,55180,-111255,78537,-117015,-89121,0
C00850=35549,55017,-111754,78289,-116991,-89291,0
C00851=36109,54738,-112612,77608,-117064,-89611,0
C00852=34833,55237,-111074,57303,-126223,-92028,0
C00853=36920,53496,-116491,54075,-124747,-93803,0
C00854=39301,53511,-116497,73795,-117548,-91141,0
C00855=44190,56115,-108651,69773,-122145,-89499,0
C00856=34852,55219,-111129,79078,-116782,-89028,0
C00857=32962,57163,-105361,81674,-116987,-87099,0
C00858=36072,54267,-114059,77471,-116694,-90045,0
C00859=40137,51524,-123057,72109,-115961,-93229,0
C00860=48403,53017,-118302,63789,-120767,-92862,0
C00861=48426,53032,-118256,63772,-120792,-92852,0
C00862=48501,53076,-118115,63710,-120874,-92824,0
C00863=48570,53109,-118011,63650,-120939,-92804,0
C00864=48660,53145,-117898,63568,-121016,-92786,0
C00865=48738,53169,-117821,63495,-121076,-92776,0
C00866=48840,53196,-117738,63395,-121147,-92768,0
C00867=48922,53212,-117688,63314,-121197,-92767,0
C00868=49032,53228,-117641,63200,-121258,-92770,0
C00869=49115,53235,-117621,63113,-121299,-92777,0
C00870=49231,53239,-117610,62988,-121347,-92791,0
C00871=49298,53238,-117615,62914,-121373,-92802,0
C00872=49408,53234,-117632,62791,-121408,-92824,0
C00873=49503,53224,-117665,62682,-121434,-92848,0
C00874=49597,53211,-117709,62573,-121453,-92874,0
C00875=49687,53192,-117774,62465,-121463,-92905,0
C00876=49775,53170,-117847,62358,-121470,-92939,0
C00877=49856,53142,-117939,62256,-121466,-92977,0
C00878=49933,53111,-118040,62156,-121458,-93017,0
C00879=49956,53100,-118078,62126,-121452,-93031,0
C00880=50003,53076,-118157,62063,-121439,-93060,0
C00881=50067,53038,-118281,61973,-121416,-93104,0
C00882=50122,52996,-118419,61893,-121384,-93150,0
C00883=50171,52952,-118562,61818,-121347,-93197,0
C00884=50185,52936,-118614,61795,-121332,-93214,0
C00885=50231,52874,-118816,61715,-121272,-93277,0
C00886=50249,52841,-118926,61679,-121236,-93310,0
C00887=50262,52808,-119032,61650,-121200,-93341,0
C00888=50275,52759,-119195,61612,-121142,-93388,0
C00889=50278,52701,-119381,61582,-121069,-93440,0
C00890=50276,52666,-119496,61567,-121024,-93472,0
C00891=50268,52633,-119606,61560,-120977,-93501,0
C00892=50258,52599,-119719,61554,-120930,-93531,0
C00893=50243,52565,-119827,61555,-120882,-93559,0
C00894=50222,52534,-119929,61563,-120835,-93584,0
C00895=50197,52499,-120044,61574,-120781,-93612,0
C00896=50170,52469,-120142,61590,-120733,-93635,0
C00897=50138,52441,-120234,61612,-120684,-93656,0
C00898=50097,52408,-120344,61641,-120627,-93681,0
C00899=50060,52382,-120429,61670,-120580,-93699,0
C00900=50018,52358,-120507,61705,-120534,-93715,0
C00901=49961,52327,-120607,61754,-120474,-93735,0
C00902=49915,52306,-120676,61794,-120430,-93747,0
C00903=49865,52287,-120738,61840,-120389,-93757,0
C00904=49793,52261,-120822,61908,-120329,-93771,0
C00905=49741,52246,-120873,61958,-120291,-93777,0
C00906=49685,52232,-120916,62013,-120253,-93782,0
C00907=49600,52213,-120979,62098,-120199,-93786,0
C00908=49545,52203,-121011,62154,-120167,-93787,0
C00909=49486,52195,-121035,62216,-120136,-93786,0
C00910=49412,52186,-121062,62293,-120098,-93783,0
C00911=49333,52180,-121082,62376,-120063,-93777,0
C00912=49219,52176,-121090,62501,-120018,-93764,0
C00913=49171,52176,-121089,62554,-120002,-93757,0
C00914=49116,52177,-121084,62615,-119983,-93748,0
C00915=49057,52181,-121069,62681,-119968,-93735,0
C00916=48978,52187,-121046,62772,-119948,-93718,0
C00917=48901,52196,-121015,62860,-119932,-93698,0
C00918=48795,52215,-120950,62986,-119919,-93665,0
C00919=48697,52238,-120868,63104,-119914,-93628,0
C00920=48607,52268,-120766,63216,-119920,-93587,0
C00921=48522,52300,-120656,63325,-119930,-93543,0
C00922=48504,52309,-120626,63349,-119935,-93533,0
C00923=48446,52339,-120527,63426,-119952,-93496,0
C00924=48376,52379,-120390,63521,-119978,-93448,0
C00925=48318,52424,-120240,63606,-120012,-93397,0
C00926=48266,52471,-120082,63685,-120052,-93345,0
C00927=48228,52522,-119916,63750,-120099,-93292,0
C00928=48218,52538,-119860,63769,-120117,-93276,0
C00929=48200,52574,-119743,63805,-120153,-93240,0
C00930=48191,52601,-119651,63828,-120184,-93212,0
C00931=48186,52627,-119566,63845,-120214,-93187,0
C00932=48180,52684,-119381,63878,-120281,-93135,0
C00933=48185,52723,-119252,63891,-120330,-93099,0
C00934=48195,52762,-119125,63898,-120382,-93064,0
C00935=48204,52792,-119027,63903,-120421,-93038,0
C00936=48217,52820,-118938,63901,-120459,-93014,0
C00937=48230,52842,-118868,63897,-120490,-92996,0
C00938=48267,52896,-118691,63881,-120571,-92952,0
C00939=48301,52933,-118574,63861,-120627,-92924,0
C00940=48337,52965,-118470,63837,-120679,-92900,0
C00941=48346,52973,-118442,63831,-120692,-92893,0
C00942=48369,53023,-118285,63829,-120760,-92852,0
C00943=30446,51903,-121560,60508,-120292,-94081,0
C00944=30471,51879,-121640,60469,-120268,-94107,0
C00945=30490,51857,-121714,60439,-120245,-94130,0
C00946=30527,51805,-121890,60373,-120187,-94184,0
C00947=30548,51762,-122035,60330,-120135,-94227,0
C00948=30563,51708,-122221,60288,-120065,-94281,0
C00949=30565,51666,-122364,60266,-120006,-94321,0
C00950=30557,51610,-122553,60249,-119927,-94372,0
C00951=30542,51570,-122690,60247,-119866,-94408,0
C00952=30509,51516,-122873,60258,-119779,-94454,0
C00953=30484,51486,-122977,60272,-119728,-94479,0
C00954=30437,51437,-123145,60302,-119643,-94519,0
C00955=30385,51396,-123284,60341,-119568,-94550,0
C00956=30327,51357,-123416,60387,-119495,-94579,0
C00957=30258,51322,-123535,60447,-119423,-94603,0
C00958=30184,51289,-123649,60513,-119351,-94625,0
C00959=30101,51261,-123745,60592,-119285,-94640,0
C00960=30014,51235,-123832,60676,-119219,-94653,0
C00961=29983,51228,-123857,60708,-119198,-94655,0
C00962=29921,51215,-123902,60771,-119159,-94659,0
C00963=29824,51197,-123961,60869,-119103,-94664,0
C00964=29723,51186,-124000,60976,-119054,-94661,0
C00965=29620,51177,-124028,61085,-119008,-94655,0
C00966=29585,51176,-124032,61124,-118995,-94651,0
C00967=29448,51174,-124035,61274,-118948,-94634,0
C00968=29377,51176,-124025,61354,-118927,-94621,0
C00969=29310,51181,-124009,61430,-118912,-94608,0
C00970=29208,51190,-123973,61546,-118892,-94585,0
C00971=29097,51207,-123915,61676,-118878,-94553,0
C00972=29030,51219,-123872,61756,-118872,-94532,0
C00973=28967,51233,-123822,61831,-118871,-94509,0
C00974=28905,51248,-123769,61907,-118871,-94486,0
C00975=28846,51265,-123708,61979,-118876,-94461,0
C00976=28793,51284,-123642,62046,-118884,-94435,0
C00977=28735,51306,-123564,62120,-118895,-94405,0
C00978=28688,51327,-123489,62182,-118908,-94378,0
C00979=28645,51350,-123409,62239,-118925,-94350,0
C00980=28595,51378,-123310,62307,-118948,-94315,0
C00981=28559,51403,-123224,62358,-118969,-94286,0
C00982=28528,51429,-123134,62403,-118994,-94256,0
C00983=28490,51464,-123014,62461,-119027,-94217,0
C00984=28467,51491,-122921,62499,-119056,-94187,0
C00985=28449,51519,-122825,62532,-119087,-94158,0
C00986=28426,51559,-122687,62575,-119133,-94115,0
C00987=28415,51587,-122592,62600,-119166,-94087,0
C00988=28410,51616,-122493,62619,-119203,-94058,0
C00989=28404,51660,-122344,62645,-119259,-94015,0
//INST
///DATE 2025/02/20 16:20
///COMM Generated using RoboDK
///ATTR SC,RW
///GROUP1 RB1
NOP
MOVL C00000 V=30.0 PL=1
MOVL C00001 V=30.0 PL=1
MOVL C00002 V=30.0 PL=1
MOVL C00003 V=30.0 PL=1
MOVL C00004 V=30.0 PL=1
MOVL C00005 V=30.0 PL=1
MOVL C00006 V=30.0 PL=1
MOVL C00007 V=30.0 PL=1
MOVL C00008 V=30.0 PL=1
MOVL C00009 V=30.0 PL=1
MOVL C00010 V=30.0 PL=1
MOVL C00011 V=30.0 PL=1
MOVL C00012 V=30.0 PL=1
MOVL C00013 V=30.0 PL=1
MOVL C00014 V=30.0 PL=1
MOVL C00015 V=30.0 PL=1
MOVL C00016 V=30.0 PL=1
MOVL C00017 V=30.0 PL=1
MOVL C00018 V=30.0 PL=1
MOVL C00019 V=30.0 PL=1
MOVL C00020 V=30.0 PL=1
MOVL C00021 V=30.0 PL=1
MOVL C00022 V=30.0 PL=1
MOVL C00023 V=30.0 PL=1
MOVL C00024 V=30.0 PL=1
MOVL C00025 V=30.0 PL=1
MOVL C00026 V=30.0 PL=1
MOVL C00027 V=30.0 PL=1
MOVL C00028 V=30.0 PL=1
MOVL C00029 V=30.0 PL=1
MOVL C00030 V=30.0 PL=1
MOVL C00031 V=30.0 PL=1
MOVL C00032 V=30.0 PL=1
MOVL C00033 V=30.0 PL=1
MOVL C00034 V=30.0 PL=1
MOVL C00035 V=30.0 PL=1
MOVL C00036 V=30.0 PL=1
MOVL C00037 V=30.0 PL=1
MOVL C00038 V=30.0 PL=1
MOVL C00039 V=30.0 PL=1
MOVL C00040 V=30.0 PL=1
MOVL C00041 V=30.0 PL=1
MOVL C00042 V=30.0 PL=1
MOVL C00043 V=30.0 PL=1
MOVL C00044 V=30.0 PL=1
MOVL C00045 V=30.0 PL=1
MOVL C00046 V=30.0 PL=1
MOVL C00047 V=30.0 PL=1
MOVL C00048 V=30.0 PL=1
MOVL C00049 V=30.0 PL=1
MOVL C00050 V=30.0 PL=1
MOVL C00051 V=30.0 PL=1
MOVL C00052 V=30.0 PL=1
MOVL C00053 V=30.0 PL=1
MOVL C00054 V=30.0 PL=1
MOVL C00055 V=30.0 PL=1
MOVL C00056 V=30.0 PL=1
MOVL C00057 V=30.0 PL=1
MOVL C00058 V=30.0 PL=1
MOVL C00059 V=30.0 PL=1
MOVL C00060 V=30.0 PL=1
MOVL C00061 V=30.0 PL=1
MOVL C00062 V=30.0 PL=1
MOVL C00063 V=30.0 PL=1
MOVL C00064 V=30.0 PL=1
MOVL C00065 V=30.0 PL=1
MOVL C00066 V=30.0 PL=1
MOVL C00067 V=30.0 PL=1
MOVL C00068 V=30.0 PL=1
MOVL C00069 V=30.0 PL=1
MOVL C00070 V=30.0 PL=1
MOVL C00071 V=30.0 PL=1
MOVL C00072 V=30.0 PL=1
MOVL C00073 V=30.0 PL=1
MOVL C00074 V=130.0 PL=1
MOVL C00075 V=130.0 PL=1
MOVL C00076 V=30.0 PL=1
MOVL C00077 V=130.0 PL=1
MOVL C00078 V=130.0 PL=1
MOVL C00079 V=30.0 PL=1
MOVL C00080 V=30.0 PL=1
MOVL C00081 V=30.0 PL=1
MOVL C00082 V=30.0 PL=1
MOVL C00083 V=30.0 PL=1
MOVL C00084 V=30.0 PL=1
MOVL C00085 V=30.0 PL=1
MOVL C00086 V=30.0 PL=1
MOVL C00087 V=30.0 PL=1
MOVL C00088 V=30.0 PL=1
MOVL C00089 V=30.0 PL=1
MOVL C00090 V=30.0 PL=1
MOVL C00091 V=30.0 PL=1
MOVL C00092 V=30.0 PL=1
MOVL C00093 V=30.0 PL=1
MOVL C00094 V=30.0 PL=1
MOVL C00095 V=30.0 PL=1
MOVL C00096 V=30.0 PL=1
MOVL C00097 V=30.0 PL=1
MOVL C00098 V=30.0 PL=1
MOVL C00099 V=30.0 PL=1
MOVL C00100 V=30.0 PL=1
MOVL C00101 V=30.0 PL=1
MOVL C00102 V=30.0 PL=1
MOVL C00103 V=30.0 PL=1
MOVL C00104 V=30.0 PL=1
MOVL C00105 V=30.0 PL=1
MOVL C00106 V=30.0 PL=1
MOVL C00107 V=30.0 PL=1
MOVL C00108 V=30.0 PL=1
MOVL C00109 V=30.0 PL=1
MOVL C00110 V=30.0 PL=1
MOVL C00111 V=30.0 PL=1
MOVL C00112 V=30.0 PL=1
MOVL C00113 V=30.0 PL=1
MOVL C00114 V=30.0 PL=1
MOVL C00115 V=30.0 PL=1
MOVL C00116 V=30.0 PL=1
MOVL C00117 V=30.0 PL=1
MOVL C00118 V=30.0 PL=1
MOVL C00119 V=30.0 PL=1
MOVL C00120 V=30.0 PL=1
MOVL C00121 V=30.0 PL=1
MOVL C00122 V=30.0 PL=1
MOVL C00123 V=30.0 PL=1
MOVL C00124 V=30.0 PL=1
MOVL C00125 V=30.0 PL=1
MOVL C00126 V=30.0 PL=1
MOVL C00127 V=30.0 PL=1
MOVL C00128 V=30.0 PL=1
MOVL C00129 V=30.0 PL=1
MOVL C00130 V=30.0 PL=1
MOVL C00131 V=30.0 PL=1
MOVL C00132 V=30.0 PL=1
MOVL C00133 V=30.0 PL=1
MOVL C00134 V=30.0 PL=1
MOVL C00135 V=30.0 PL=1
MOVL C00136 V=30.0 PL=1
MOVL C00137 V=30.0 PL=1
MOVL C00138 V=30.0 PL=1
MOVL C00139 V=30.0 PL=1
MOVL C00140 V=30.0 PL=1
MOVL C00141 V=30.0 PL=1
MOVL C00142 V=30.0 PL=1
MOVL C00143 V=30.0 PL=1
MOVL C00144 V=30.0 PL=1
MOVL C00145 V=30.0 PL=1
MOVL C00146 V=30.0 PL=1
MOVL C00147 V=30.0 PL=1
MOVL C00148 V=30.0 PL=1
MOVL C00149 V=30.0 PL=1
MOVL C00150 V=30.0 PL=1
MOVL C00151 V=30.0 PL=1
MOVL C00152 V=30.0 PL=1
MOVL C00153 V=130.0 PL=1
MOVL C00154 V=130.0 PL=1
MOVL C00155 V=60.0 PL=1
MOVL C00156 V=60.0 PL=1
MOVL C00157 V=60.0 PL=1
MOVL C00158 V=60.0 PL=1
MOVL C00159 V=130.0 PL=1
MOVL C00160 V=30.0 PL=1
MOVL C00161 V=30.0 PL=1
MOVL C00162 V=30.0 PL=1
MOVL C00163 V=30.0 PL=1
MOVL C00164 V=30.0 PL=1
MOVL C00165 V=30.0 PL=1
MOVL C00166 V=30.0 PL=1
MOVL C00167 V=30.0 PL=1
MOVL C00168 V=130.0 PL=1
MOVL C00169 V=130.0 PL=1
MOVL C00170 V=30.0 PL=1
MOVL C00171 V=130.0 PL=1
MOVL C00172 V=30.0 PL=1
MOVL C00173 V=130.0 PL=1
MOVL C00174 V=30.0 PL=1
MOVL C00175 V=130.0 PL=1
MOVL C00176 V=20.0 PL=1
MOVL C00177 V=130.0 PL=1
MOVL C00178 V=30.0 PL=1
MOVL C00179 V=30.0 PL=1
MOVL C00180 V=30.0 PL=1
MOVL C00181 V=30.0 PL=1
MOVL C00182 V=30.0 PL=1
MOVL C00183 V=30.0 PL=1
MOVL C00184 V=30.0 PL=1
MOVL C00185 V=30.0 PL=1
MOVL C00186 V=30.0 PL=1
MOVL C00187 V=30.0 PL=1
MOVL C00188 V=30.0 PL=1
MOVL C00189 V=30.0 PL=1
MOVL C00190 V=30.0 PL=1
MOVL C00191 V=30.0 PL=1
MOVL C00192 V=30.0 PL=1
MOVL C00193 V=30.0 PL=1
MOVL C00194 V=30.0 PL=1
MOVL C00195 V=30.0 PL=1
MOVL C00196 V=30.0 PL=1
MOVL C00197 V=30.0 PL=1
MOVL C00198 V=30.0 PL=1
MOVL C00199 V=30.0 PL=1
MOVL C00200 V=30.0 PL=1
MOVL C00201 V=30.0 PL=1
MOVL C00202 V=30.0 PL=1
MOVL C00203 V=30.0 PL=1
MOVL C00204 V=30.0 PL=1
MOVL C00205 V=30.0 PL=1
MOVL C00206 V=30.0 PL=1
MOVL C00207 V=30.0 PL=1
MOVL C00208 V=30.0 PL=1
MOVL C00209 V=30.0 PL=1
MOVL C00210 V=30.0 PL=1
MOVL C00211 V=30.0 PL=1
MOVL C00212 V=30.0 PL=1
MOVL C00213 V=30.0 PL=1
MOVL C00214 V=30.0 PL=1
MOVL C00215 V=30.0 PL=1
MOVL C00216 V=30.0 PL=1
MOVL C00217 V=30.0 PL=1
MOVL C00218 V=30.0 PL=1
MOVL C00219 V=30.0 PL=1
MOVL C00220 V=30.0 PL=1
MOVL C00221 V=30.0 PL=1
MOVL C00222 V=30.0 PL=1
MOVL C00223 V=30.0 PL=1
MOVL C00224 V=30.0 PL=1
MOVL C00225 V=30.0 PL=1
MOVL C00226 V=30.0 PL=1
MOVL C00227 V=30.0 PL=1
MOVL C00228 V=30.0 PL=1
MOVL C00229 V=30.0 PL=1
MOVL C00230 V=30.0 PL=1
MOVL C00231 V=30.0 PL=1
MOVL C00232 V=30.0 PL=1
MOVL C00233 V=30.0 PL=1
MOVL C00234 V=30.0 PL=1
MOVL C00235 V=30.0 PL=1
MOVL C00236 V=30.0 PL=1
MOVL C00237 V=30.0 PL=1
MOVL C00238 V=30.0 PL=1
MOVL C00239 V=30.0 PL=1
MOVL C00240 V=30.0 PL=1
MOVL C00241 V=30.0 PL=1
MOVL C00242 V=30.0 PL=1
MOVL C00243 V=30.0 PL=1
MOVL C00244 V=30.0 PL=1
MOVL C00245 V=30.0 PL=1
MOVL C00246 V=30.0 PL=1
MOVL C00247 V=30.0 PL=1
MOVL C00248 V=30.0 PL=1
MOVL C00249 V=30.0 PL=1
MOVL C00250 V=30.0 PL=1
MOVL C00251 V=130.0 PL=1
MOVL C00252 V=130.0 PL=1
MOVL C00253 V=30.0 PL=1
MOVL C00254 V=30.0 PL=1
MOVL C00255 V=30.0 PL=1
MOVL C00256 V=30.0 PL=1
MOVL C00257 V=30.0 PL=1
MOVL C00258 V=30.0 PL=1
MOVL C00259 V=30.0 PL=1
MOVL C00260 V=30.0 PL=1
MOVL C00261 V=30.0 PL=1
MOVL C00262 V=30.0 PL=1
MOVL C00263 V=30.0 PL=1
MOVL C00264 V=30.0 PL=1
MOVL C00265 V=30.0 PL=1
MOVL C00266 V=30.0 PL=1
MOVL C00267 V=30.0 PL=1
MOVL C00268 V=30.0 PL=1
MOVL C00269 V=30.0 PL=1
MOVL C00270 V=30.0 PL=1
MOVL C00271 V=30.0 PL=1
MOVL C00272 V=30.0 PL=1
MOVL C00273 V=30.0 PL=1
MOVL C00274 V=30.0 PL=1
MOVL C00275 V=30.0 PL=1
MOVL C00276 V=30.0 PL=1
MOVL C00277 V=30.0 PL=1
MOVL C00278 V=30.0 PL=1
MOVL C00279 V=30.0 PL=1
MOVL C00280 V=30.0 PL=1
MOVL C00281 V=30.0 PL=1
MOVL C00282 V=30.0 PL=1
MOVL C00283 V=30.0 PL=1
MOVL C00284 V=30.0 PL=1
MOVL C00285 V=30.0 PL=1
MOVL C00286 V=30.0 PL=1
MOVL C00287 V=30.0 PL=1
MOVL C00288 V=30.0 PL=1
MOVL C00289 V=30.0 PL=1
MOVL C00290 V=30.0 PL=1
MOVL C00291 V=30.0 PL=1
MOVL C00292 V=30.0 PL=1
MOVL C00293 V=30.0 PL=1
MOVL C00294 V=30.0 PL=1
MOVL C00295 V=30.0 PL=1
MOVL C00296 V=30.0 PL=1
MOVL C00297 V=30.0 PL=1
MOVL C00298 V=30.0 PL=1
MOVL C00299 V=30.0 PL=1
MOVL C00300 V=30.0 PL=1
MOVL C00301 V=30.0 PL=1
MOVL C00302 V=30.0 PL=1
MOVL C00303 V=30.0 PL=1
MOVL C00304 V=30.0 PL=1
MOVL C00305 V=30.0 PL=1
MOVL C00306 V=30.0 PL=1
MOVL C00307 V=30.0 PL=1
MOVL C00308 V=30.0 PL=1
MOVL C00309 V=30.0 PL=1
MOVL C00310 V=30.0 PL=1
MOVL C00311 V=30.0 PL=1
MOVL C00312 V=30.0 PL=1
MOVL C00313 V=30.0 PL=1
MOVL C00314 V=30.0 PL=1
MOVL C00315 V=30.0 PL=1
MOVL C00316 V=30.0 PL=1
MOVL C00317 V=30.0 PL=1
MOVL C00318 V=30.0 PL=1
MOVL C00319 V=30.0 PL=1
MOVL C00320 V=30.0 PL=1
MOVL C00321 V=30.0 PL=1
MOVL C00322 V=30.0 PL=1
MOVL C00323 V=30.0 PL=1
MOVL C00324 V=30.0 PL=1
MOVL C00325 V=30.0 PL=1
MOVL C00326 V=30.0 PL=1
MOVL C00327 V=30.0 PL=1
MOVL C00328 V=30.0 PL=1
MOVL C00329 V=130.0 PL=1
MOVL C00330 V=130.0 PL=1
MOVL C00331 V=30.0 PL=1
MOVL C00332 V=130.0 PL=1
MOVL C00333 V=30.0 PL=1
MOVL C00334 V=30.0 PL=1
MOVL C00335 V=30.0 PL=1
MOVL C00336 V=30.0 PL=1
MOVL C00337 V=30.0 PL=1
MOVL C00338 V=30.0 PL=1
MOVL C00339 V=30.0 PL=1
MOVL C00340 V=30.0 PL=1
MOVL C00341 V=30.0 PL=1
MOVL C00342 V=30.0 PL=1
MOVL C00343 V=30.0 PL=1
MOVL C00344 V=30.0 PL=1
MOVL C00345 V=30.0 PL=1
MOVL C00346 V=30.0 PL=1
MOVL C00347 V=30.0 PL=1
MOVL C00348 V=30.0 PL=1
MOVL C00349 V=30.0 PL=1
MOVL C00350 V=30.0 PL=1
MOVL C00351 V=30.0 PL=1
MOVL C00352 V=30.0 PL=1
MOVL C00353 V=30.0 PL=1
MOVL C00354 V=30.0 PL=1
MOVL C00355 V=30.0 PL=1
MOVL C00356 V=30.0 PL=1
MOVL C00357 V=30.0 PL=1
MOVL C00358 V=30.0 PL=1
MOVL C00359 V=30.0 PL=1
MOVL C00360 V=30.0 PL=1
MOVL C00361 V=30.0 PL=1
MOVL C00362 V=30.0 PL=1
MOVL C00363 V=30.0 PL=1
MOVL C00364 V=30.0 PL=1
MOVL C00365 V=30.0 PL=1
MOVL C00366 V=30.0 PL=1
MOVL C00367 V=30.0 PL=1
MOVL C00368 V=30.0 PL=1
MOVL C00369 V=30.0 PL=1
MOVL C00370 V=30.0 PL=1
MOVL C00371 V=30.0 PL=1
MOVL C00372 V=30.0 PL=1
MOVL C00373 V=30.0 PL=1
MOVL C00374 V=30.0 PL=1
MOVL C00375 V=30.0 PL=1
MOVL C00376 V=30.0 PL=1
MOVL C00377 V=30.0 PL=1
MOVL C00378 V=30.0 PL=1
MOVL C00379 V=30.0 PL=1
MOVL C00380 V=30.0 PL=1
MOVL C00381 V=30.0 PL=1
MOVL C00382 V=30.0 PL=1
MOVL C00383 V=30.0 PL=1
MOVL C00384 V=30.0 PL=1
MOVL C00385 V=30.0 PL=1
MOVL C00386 V=30.0 PL=1
MOVL C00387 V=30.0 PL=1
MOVL C00388 V=30.0 PL=1
MOVL C00389 V=30.0 PL=1
MOVL C00390 V=30.0 PL=1
MOVL C00391 V=30.0 PL=1
MOVL C00392 V=30.0 PL=1
MOVL C00393 V=30.0 PL=1
MOVL C00394 V=30.0 PL=1
MOVL C00395 V=30.0 PL=1
MOVL C00396 V=30.0 PL=1
MOVL C00397 V=30.0 PL=1
MOVL C00398 V=30.0 PL=1
MOVL C00399 V=30.0 PL=1
MOVL C00400 V=30.0 PL=1
MOVL C00401 V=30.0 PL=1
MOVL C00402 V=30.0 PL=1
MOVL C00403 V=30.0 PL=1
MOVL C00404 V=30.0 PL=1
MOVL C00405 V=30.0 PL=1
MOVL C00406 V=30.0 PL=1
MOVL C00407 V=130.0 PL=1
MOVL C00408 V=130.0 PL=1
MOVL C00409 V=130.0 PL=1
MOVL C00410 V=30.0 PL=1
MOVL C00411 V=30.0 PL=1
MOVL C00412 V=30.0 PL=1
MOVL C00413 V=30.0 PL=1
MOVL C00414 V=30.0 PL=1
MOVL C00415 V=30.0 PL=1
MOVL C00416 V=30.0 PL=1
MOVL C00417 V=30.0 PL=1
MOVL C00418 V=30.0 PL=1
MOVL C00419 V=30.0 PL=1
MOVL C00420 V=30.0 PL=1
MOVL C00421 V=30.0 PL=1
MOVL C00422 V=30.0 PL=1
MOVL C00423 V=30.0 PL=1
MOVL C00424 V=30.0 PL=1
MOVL C00425 V=30.0 PL=1
MOVL C00426 V=30.0 PL=1
MOVL C00427 V=30.0 PL=1
MOVL C00428 V=30.0 PL=1
MOVL C00429 V=30.0 PL=1
MOVL C00430 V=30.0 PL=1
MOVL C00431 V=30.0 PL=1
MOVL C00432 V=30.0 PL=1
MOVL C00433 V=30.0 PL=1
MOVL C00434 V=30.0 PL=1
MOVL C00435 V=30.0 PL=1
MOVL C00436 V=30.0 PL=1
MOVL C00437 V=30.0 PL=1
MOVL C00438 V=30.0 PL=1
MOVL C00439 V=30.0 PL=1
MOVL C00440 V=30.0 PL=1
MOVL C00441 V=30.0 PL=1
MOVL C00442 V=30.0 PL=1
MOVL C00443 V=30.0 PL=1
MOVL C00444 V=30.0 PL=1
MOVL C00445 V=30.0 PL=1
MOVL C00446 V=30.0 PL=1
MOVL C00447 V=30.0 PL=1
MOVL C00448 V=30.0 PL=1
MOVL C00449 V=30.0 PL=1
MOVL C00450 V=30.0 PL=1
MOVL C00451 V=30.0 PL=1
MOVL C00452 V=30.0 PL=1
MOVL C00453 V=30.0 PL=1
MOVL C00454 V=30.0 PL=1
MOVL C00455 V=30.0 PL=1
MOVL C00456 V=30.0 PL=1
MOVL C00457 V=30.0 PL=1
MOVL C00458 V=30.0 PL=1
MOVL C00459 V=30.0 PL=1
MOVL C00460 V=30.0 PL=1
MOVL C00461 V=30.0 PL=1
MOVL C00462 V=30.0 PL=1
MOVL C00463 V=30.0 PL=1
MOVL C00464 V=30.0 PL=1
MOVL C00465 V=30.0 PL=1
MOVL C00466 V=30.0 PL=1
MOVL C00467 V=30.0 PL=1
MOVL C00468 V=30.0 PL=1
MOVL C00469 V=30.0 PL=1
MOVL C00470 V=30.0 PL=1
MOVL C00471 V=30.0 PL=1
MOVL C00472 V=30.0 PL=1
MOVL C00473 V=30.0 PL=1
MOVL C00474 V=30.0 PL=1
MOVL C00475 V=30.0 PL=1
MOVL C00476 V=30.0 PL=1
MOVL C00477 V=30.0 PL=1
MOVL C00478 V=30.0 PL=1
MOVL C00479 V=30.0 PL=1
MOVL C00480 V=30.0 PL=1
MOVL C00481 V=30.0 PL=1
MOVL C00482 V=30.0 PL=1
MOVL C00483 V=30.0 PL=1
MOVL C00484 V=30.0 PL=1
MOVL C00485 V=30.0 PL=1
MOVL C00486 V=30.0 PL=1
MOVL C00487 V=30.0 PL=1
MOVL C00488 V=130.0 PL=1
MOVL C00489 V=130.0 PL=1
MOVL C00490 V=60.0 PL=1
MOVL C00491 V=60.0 PL=1
MOVL C00492 V=60.0 PL=1
MOVL C00493 V=60.0 PL=1
MOVL C00494 V=130.0 PL=1
MOVL C00495 V=30.0 PL=1
MOVL C00496 V=30.0 PL=1
MOVL C00497 V=30.0 PL=1
MOVL C00498 V=30.0 PL=1
MOVL C00499 V=30.0 PL=1
MOVL C00500 V=30.0 PL=1
MOVL C00501 V=30.0 PL=1
MOVL C00502 V=30.0 PL=1
MOVL C00503 V=130.0 PL=1
MOVL C00504 V=130.0 PL=1
MOVL C00505 V=30.0 PL=1
MOVL C00506 V=130.0 PL=1
MOVL C00507 V=30.0 PL=1
MOVL C00508 V=130.0 PL=1
MOVL C00509 V=30.0 PL=1
MOVL C00510 V=130.0 PL=1
MOVL C00511 V=20.0 PL=1
MOVL C00512 V=130.0 PL=1
MOVL C00513 V=30.0 PL=1
MOVL C00514 V=30.0 PL=1
MOVL C00515 V=30.0 PL=1
MOVL C00516 V=30.0 PL=1
MOVL C00517 V=30.0 PL=1
MOVL C00518 V=30.0 PL=1
MOVL C00519 V=30.0 PL=1
MOVL C00520 V=30.0 PL=1
MOVL C00521 V=30.0 PL=1
MOVL C00522 V=30.0 PL=1
MOVL C00523 V=30.0 PL=1
MOVL C00524 V=30.0 PL=1
MOVL C00525 V=30.0 PL=1
MOVL C00526 V=30.0 PL=1
MOVL C00527 V=30.0 PL=1
MOVL C00528 V=30.0 PL=1
MOVL C00529 V=30.0 PL=1
MOVL C00530 V=30.0 PL=1
MOVL C00531 V=30.0 PL=1
MOVL C00532 V=30.0 PL=1
MOVL C00533 V=30.0 PL=1
MOVL C00534 V=30.0 PL=1
MOVL C00535 V=30.0 PL=1
MOVL C00536 V=30.0 PL=1
MOVL C00537 V=30.0 PL=1
MOVL C00538 V=30.0 PL=1
MOVL C00539 V=30.0 PL=1
MOVL C00540 V=30.0 PL=1
MOVL C00541 V=30.0 PL=1
MOVL C00542 V=30.0 PL=1
MOVL C00543 V=30.0 PL=1
MOVL C00544 V=30.0 PL=1
MOVL C00545 V=30.0 PL=1
MOVL C00546 V=30.0 PL=1
MOVL C00547 V=30.0 PL=1
MOVL C00548 V=30.0 PL=1
MOVL C00549 V=30.0 PL=1
MOVL C00550 V=30.0 PL=1
MOVL C00551 V=30.0 PL=1
MOVL C00552 V=30.0 PL=1
MOVL C00553 V=30.0 PL=1
MOVL C00554 V=30.0 PL=1
MOVL C00555 V=30.0 PL=1
MOVL C00556 V=30.0 PL=1
MOVL C00557 V=30.0 PL=1
MOVL C00558 V=30.0 PL=1
MOVL C00559 V=30.0 PL=1
MOVL C00560 V=30.0 PL=1
MOVL C00561 V=30.0 PL=1
MOVL C00562 V=30.0 PL=1
MOVL C00563 V=30.0 PL=1
MOVL C00564 V=30.0 PL=1
MOVL C00565 V=30.0 PL=1
MOVL C00566 V=30.0 PL=1
MOVL C00567 V=30.0 PL=1
MOVL C00568 V=30.0 PL=1
MOVL C00569 V=30.0 PL=1
MOVL C00570 V=30.0 PL=1
MOVL C00571 V=30.0 PL=1
MOVL C00572 V=30.0 PL=1
MOVL C00573 V=30.0 PL=1
MOVL C00574 V=30.0 PL=1
MOVL C00575 V=30.0 PL=1
MOVL C00576 V=30.0 PL=1
MOVL C00577 V=30.0 PL=1
MOVL C00578 V=30.0 PL=1
MOVL C00579 V=30.0 PL=1
MOVL C00580 V=30.0 PL=1
MOVL C00581 V=30.0 PL=1
MOVL C00582 V=30.0 PL=1
MOVL C00583 V=30.0 PL=1
MOVL C00584 V=30.0 PL=1
MOVL C00585 V=30.0 PL=1
MOVL C00586 V=30.0 PL=1
MOVL C00587 V=30.0 PL=1
MOVL C00588 V=30.0 PL=1
MOVL C00589 V=30.0 PL=1
MOVL C00590 V=130.0 PL=1
MOVL C00591 V=130.0 PL=1
MOVL C00592 V=30.0 PL=1
MOVL C00593 V=30.0 PL=1
MOVL C00594 V=30.0 PL=1
MOVL C00595 V=30.0 PL=1
MOVL C00596 V=30.0 PL=1
MOVL C00597 V=30.0 PL=1
MOVL C00598 V=30.0 PL=1
MOVL C00599 V=30.0 PL=1
MOVL C00600 V=30.0 PL=1
MOVL C00601 V=30.0 PL=1
MOVL C00602 V=30.0 PL=1
MOVL C00603 V=30.0 PL=1
MOVL C00604 V=30.0 PL=1
MOVL C00605 V=30.0 PL=1
MOVL C00606 V=30.0 PL=1
MOVL C00607 V=30.0 PL=1
MOVL C00608 V=30.0 PL=1
MOVL C00609 V=30.0 PL=1
MOVL C00610 V=30.0 PL=1
MOVL C00611 V=30.0 PL=1
MOVL C00612 V=30.0 PL=1
MOVL C00613 V=30.0 PL=1
MOVL C00614 V=30.0 PL=1
MOVL C00615 V=30.0 PL=1
MOVL C00616 V=30.0 PL=1
MOVL C00617 V=30.0 PL=1
MOVL C00618 V=30.0 PL=1
MOVL C00619 V=30.0 PL=1
MOVL C00620 V=30.0 PL=1
MOVL C00621 V=30.0 PL=1
MOVL C00622 V=30.0 PL=1
MOVL C00623 V=30.0 PL=1
MOVL C00624 V=30.0 PL=1
MOVL C00625 V=30.0 PL=1
MOVL C00626 V=30.0 PL=1
MOVL C00627 V=30.0 PL=1
MOVL C00628 V=30.0 PL=1
MOVL C00629 V=30.0 PL=1
MOVL C00630 V=30.0 PL=1
MOVL C00631 V=30.0 PL=1
MOVL C00632 V=30.0 PL=1
MOVL C00633 V=30.0 PL=1
MOVL C00634 V=30.0 PL=1
MOVL C00635 V=30.0 PL=1
MOVL C00636 V=30.0 PL=1
MOVL C00637 V=30.0 PL=1
MOVL C00638 V=30.0 PL=1
MOVL C00639 V=30.0 PL=1
MOVL C00640 V=30.0 PL=1
MOVL C00641 V=30.0 PL=1
MOVL C00642 V=30.0 PL=1
MOVL C00643 V=30.0 PL=1
MOVL C00644 V=30.0 PL=1
MOVL C00645 V=30.0 PL=1
MOVL C00646 V=30.0 PL=1
MOVL C00647 V=30.0 PL=1
MOVL C00648 V=30.0 PL=1
MOVL C00649 V=30.0 PL=1
MOVL C00650 V=30.0 PL=1
MOVL C00651 V=30.0 PL=1
MOVL C00652 V=30.0 PL=1
MOVL C00653 V=30.0 PL=1
MOVL C00654 V=30.0 PL=1
MOVL C00655 V=30.0 PL=1
MOVL C00656 V=30.0 PL=1
MOVL C00657 V=30.0 PL=1
MOVL C00658 V=30.0 PL=1
MOVL C00659 V=30.0 PL=1
MOVL C00660 V=30.0 PL=1
MOVL C00661 V=30.0 PL=1
MOVL C00662 V=30.0 PL=1
MOVL C00663 V=30.0 PL=1
MOVL C00664 V=30.0 PL=1
MOVL C00665 V=30.0 PL=1
MOVL C00666 V=30.0 PL=1
MOVL C00667 V=30.0 PL=1
MOVL C00668 V=30.0 PL=1
MOVL C00669 V=30.0 PL=1
MOVL C00670 V=130.0 PL=1
MOVL C00671 V=130.0 PL=1
MOVL C00672 V=30.0 PL=1
MOVL C00673 V=130.0 PL=1
MOVL C00674 V=30.0 PL=1
MOVL C00675 V=30.0 PL=1
MOVL C00676 V=30.0 PL=1
MOVL C00677 V=30.0 PL=1
MOVL C00678 V=30.0 PL=1
MOVL C00679 V=30.0 PL=1
MOVL C00680 V=30.0 PL=1
MOVL C00681 V=30.0 PL=1
MOVL C00682 V=30.0 PL=1
MOVL C00683 V=30.0 PL=1
MOVL C00684 V=30.0 PL=1
MOVL C00685 V=30.0 PL=1
MOVL C00686 V=30.0 PL=1
MOVL C00687 V=30.0 PL=1
MOVL C00688 V=30.0 PL=1
MOVL C00689 V=30.0 PL=1
MOVL C00690 V=30.0 PL=1
MOVL C00691 V=30.0 PL=1
MOVL C00692 V=30.0 PL=1
MOVL C00693 V=30.0 PL=1
MOVL C00694 V=30.0 PL=1
MOVL C00695 V=30.0 PL=1
MOVL C00696 V=30.0 PL=1
MOVL C00697 V=30.0 PL=1
MOVL C00698 V=30.0 PL=1
MOVL C00699 V=30.0 PL=1
MOVL C00700 V=30.0 PL=1
MOVL C00701 V=30.0 PL=1
MOVL C00702 V=30.0 PL=1
MOVL C00703 V=30.0 PL=1
MOVL C00704 V=30.0 PL=1
MOVL C00705 V=30.0 PL=1
MOVL C00706 V=30.0 PL=1
MOVL C00707 V=30.0 PL=1
MOVL C00708 V=30.0 PL=1
MOVL C00709 V=30.0 PL=1
MOVL C00710 V=30.0 PL=1
MOVL C00711 V=30.0 PL=1
MOVL C00712 V=30.0 PL=1
MOVL C00713 V=30.0 PL=1
MOVL C00714 V=30.0 PL=1
MOVL C00715 V=30.0 PL=1
MOVL C00716 V=30.0 PL=1
MOVL C00717 V=30.0 PL=1
MOVL C00718 V=30.0 PL=1
MOVL C00719 V=30.0 PL=1
MOVL C00720 V=30.0 PL=1
MOVL C00721 V=30.0 PL=1
MOVL C00722 V=30.0 PL=1
MOVL C00723 V=30.0 PL=1
MOVL C00724 V=30.0 PL=1
MOVL C00725 V=30.0 PL=1
MOVL C00726 V=30.0 PL=1
MOVL C00727 V=30.0 PL=1
MOVL C00728 V=30.0 PL=1
MOVL C00729 V=30.0 PL=1
MOVL C00730 V=30.0 PL=1
MOVL C00731 V=30.0 PL=1
MOVL C00732 V=30.0 PL=1
MOVL C00733 V=30.0 PL=1
MOVL C00734 V=30.0 PL=1
MOVL C00735 V=30.0 PL=1
MOVL C00736 V=30.0 PL=1
MOVL C00737 V=30.0 PL=1
MOVL C00738 V=30.0 PL=1
MOVL C00739 V=30.0 PL=1
MOVL C00740 V=30.0 PL=1
MOVL C00741 V=30.0 PL=1
MOVL C00742 V=30.0 PL=1
MOVL C00743 V=30.0 PL=1
MOVL C00744 V=30.0 PL=1
MOVL C00745 V=30.0 PL=1
MOVL C00746 V=30.0 PL=1
MOVL C00747 V=30.0 PL=1
MOVL C00748 V=30.0 PL=1
MOVL C00749 V=30.0 PL=1
MOVL C00750 V=30.0 PL=1
MOVL C00751 V=130.0 PL=1
MOVL C00752 V=130.0 PL=1
MOVL C00753 V=130.0 PL=1
MOVL C00754 V=30.0 PL=1
MOVL C00755 V=30.0 PL=1
MOVL C00756 V=30.0 PL=1
MOVL C00757 V=30.0 PL=1
MOVL C00758 V=30.0 PL=1
MOVL C00759 V=30.0 PL=1
MOVL C00760 V=30.0 PL=1
MOVL C00761 V=30.0 PL=1
MOVL C00762 V=30.0 PL=1
MOVL C00763 V=30.0 PL=1
MOVL C00764 V=30.0 PL=1
MOVL C00765 V=30.0 PL=1
MOVL C00766 V=30.0 PL=1
MOVL C00767 V=30.0 PL=1
MOVL C00768 V=30.0 PL=1
MOVL C00769 V=30.0 PL=1
MOVL C00770 V=30.0 PL=1
MOVL C00771 V=30.0 PL=1
MOVL C00772 V=30.0 PL=1
MOVL C00773 V=30.0 PL=1
MOVL C00774 V=30.0 PL=1
MOVL C00775 V=30.0 PL=1
MOVL C00776 V=30.0 PL=1
MOVL C00777 V=30.0 PL=1
MOVL C00778 V=30.0 PL=1
MOVL C00779 V=30.0 PL=1
MOVL C00780 V=30.0 PL=1
MOVL C00781 V=30.0 PL=1
MOVL C00782 V=30.0 PL=1
MOVL C00783 V=30.0 PL=1
MOVL C00784 V=30.0 PL=1
MOVL C00785 V=30.0 PL=1
MOVL C00786 V=30.0 PL=1
MOVL C00787 V=30.0 PL=1
MOVL C00788 V=30.0 PL=1
MOVL C00789 V=30.0 PL=1
MOVL C00790 V=30.0 PL=1
MOVL C00791 V=30.0 PL=1
MOVL C00792 V=30.0 PL=1
MOVL C00793 V=30.0 PL=1
MOVL C00794 V=30.0 PL=1
MOVL C00795 V=30.0 PL=1
MOVL C00796 V=30.0 PL=1
MOVL C00797 V=30.0 PL=1
MOVL C00798 V=30.0 PL=1
MOVL C00799 V=30.0 PL=1
MOVL C00800 V=30.0 PL=1
MOVL C00801 V=30.0 PL=1
MOVL C00802 V=30.0 PL=1
MOVL C00803 V=30.0 PL=1
MOVL C00804 V=30.0 PL=1
MOVL C00805 V=30.0 PL=1
MOVL C00806 V=30.0 PL=1
MOVL C00807 V=30.0 PL=1
MOVL C00808 V=30.0 PL=1
MOVL C00809 V=30.0 PL=1
MOVL C00810 V=30.0 PL=1
MOVL C00811 V=30.0 PL=1
MOVL C00812 V=30.0 PL=1
MOVL C00813 V=30.0 PL=1
MOVL C00814 V=30.0 PL=1
MOVL C00815 V=30.0 PL=1
MOVL C00816 V=30.0 PL=1
MOVL C00817 V=30.0 PL=1
MOVL C00818 V=30.0 PL=1
MOVL C00819 V=30.0 PL=1
MOVL C00820 V=30.0 PL=1
MOVL C00821 V=30.0 PL=1
MOVL C00822 V=30.0 PL=1
MOVL C00823 V=30.0 PL=1
MOVL C00824 V=30.0 PL=1
MOVL C00825 V=30.0 PL=1
MOVL C00826 V=30.0 PL=1
MOVL C00827 V=30.0 PL=1
MOVL C00828 V=30.0 PL=1
MOVL C00829 V=30.0 PL=1
MOVL C00830 V=30.0 PL=1
MOVL C00831 V=30.0 PL=1
MOVL C00832 V=30.0 PL=1
MOVL C00833 V=30.0 PL=1
MOVL C00834 V=30.0 PL=1
MOVL C00835 V=30.0 PL=1
MOVL C00836 V=130.0 PL=1
MOVL C00837 V=130.0 PL=1
MOVL C00838 V=60.0 PL=1
MOVL C00839 V=60.0 PL=1
MOVL C00840 V=60.0 PL=1
MOVL C00841 V=60.0 PL=1
MOVL C00842 V=130.0 PL=1
MOVL C00843 V=30.0 PL=1
MOVL C00844 V=30.0 PL=1
MOVL C00845 V=30.0 PL=1
MOVL C00846 V=30.0 PL=1
MOVL C00847 V=30.0 PL=1
MOVL C00848 V=30.0 PL=1
MOVL C00849 V=30.0 PL=1
MOVL C00850 V=30.0 PL=1
MOVL C00851 V=130.0 PL=1
MOVL C00852 V=130.0 PL=1
MOVL C00853 V=30.0 PL=1
MOVL C00854 V=130.0 PL=1
MOVL C00855 V=30.0 PL=1
MOVL C00856 V=130.0 PL=1
MOVL C00857 V=30.0 PL=1
MOVL C00858 V=130.0 PL=1
MOVL C00859 V=20.0 PL=1
MOVL C00860 V=130.0 PL=1
MOVL C00861 V=30.0 PL=1
MOVL C00862 V=30.0 PL=1
MOVL C00863 V=30.0 PL=1
MOVL C00864 V=30.0 PL=1
MOVL C00865 V=30.0 PL=1
MOVL C00866 V=30.0 PL=1
MOVL C00867 V=30.0 PL=1
MOVL C00868 V=30.0 PL=1
MOVL C00869 V=30.0 PL=1
MOVL C00870 V=30.0 PL=1
MOVL C00871 V=30.0 PL=1
MOVL C00872 V=30.0 PL=1
MOVL C00873 V=30.0 PL=1
MOVL C00874 V=30.0 PL=1
MOVL C00875 V=30.0 PL=1
MOVL C00876 V=30.0 PL=1
MOVL C00877 V=30.0 PL=1
MOVL C00878 V=30.0 PL=1
MOVL C00879 V=30.0 PL=1
MOVL C00880 V=30.0 PL=1
MOVL C00881 V=30.0 PL=1
MOVL C00882 V=30.0 PL=1
MOVL C00883 V=30.0 PL=1
MOVL C00884 V=30.0 PL=1
MOVL C00885 V=30.0 PL=1
MOVL C00886 V=30.0 PL=1
MOVL C00887 V=30.0 PL=1
MOVL C00888 V=30.0 PL=1
MOVL C00889 V=30.0 PL=1
MOVL C00890 V=30.0 PL=1
MOVL C00891 V=30.0 PL=1
MOVL C00892 V=30.0 PL=1
MOVL C00893 V=30.0 PL=1
MOVL C00894 V=30.0 PL=1
MOVL C00895 V=30.0 PL=1
MOVL C00896 V=30.0 PL=1
MOVL C00897 V=30.0 PL=1
MOVL C00898 V=30.0 PL=1
MOVL C00899 V=30.0 PL=1
MOVL C00900 V=30.0 PL=1
MOVL C00901 V=30.0 PL=1
MOVL C00902 V=30.0 PL=1
MOVL C00903 V=30.0 PL=1
MOVL C00904 V=30.0 PL=1
MOVL C00905 V=30.0 PL=1
MOVL C00906 V=30.0 PL=1
MOVL C00907 V=30.0 PL=1
MOVL C00908 V=30.0 PL=1
MOVL C00909 V=30.0 PL=1
MOVL C00910 V=30.0 PL=1
MOVL C00911 V=30.0 PL=1
MOVL C00912 V=30.0 PL=1
MOVL C00913 V=30.0 PL=1
MOVL C00914 V=30.0 PL=1
MOVL C00915 V=30.0 PL=1
MOVL C00916 V=30.0 PL=1
MOVL C00917 V=30.0 PL=1
MOVL C00918 V=30.0 PL=1
MOVL C00919 V=30.0 PL=1
MOVL C00920 V=30.0 PL=1
MOVL C00921 V=30.0 PL=1
MOVL C00922 V=30.0 PL=1
MOVL C00923 V=30.0 PL=1
MOVL C00924 V=30.0 PL=1
MOVL C00925 V=30.0 PL=1
MOVL C00926 V=30.0 PL=1
MOVL C00927 V=30.0 PL=1
MOVL C00928 V=30.0 PL=1
MOVL C00929 V=30.0 PL=1
MOVL C00930 V=30.0 PL=1
MOVL C00931 V=30.0 PL=1
MOVL C00932 V=30.0 PL=1
MOVL C00933 V=30.0 PL=1
MOVL C00934 V=30.0 PL=1
MOVL C00935 V=30.0 PL=1
MOVL C00936 V=30.0 PL=1
MOVL C00937 V=30.0 PL=1
MOVL C00938 V=30.0 PL=1
MOVL C00939 V=30.0 PL=1
MOVL C00940 V=30.0 PL=1
MOVL C00941 V=30.0 PL=1
MOVL C00942 V=130.0 PL=1
MOVL C00943 V=130.0 PL=1
MOVL C00944 V=30.0 PL=1
MOVL C00945 V=30.0 PL=1
MOVL C00946 V=30.0 PL=1
MOVL C00947 V=30.0 PL=1
MOVL C00948 V=30.0 PL=1
MOVL C00949 V=30.0 PL=1
MOVL C00950 V=30.0 PL=1
MOVL C00951 V=30.0 PL=1
MOVL C00952 V=30.0 PL=1
MOVL C00953 V=30.0 PL=1
MOVL C00954 V=30.0 PL=1
MOVL C00955 V=30.0 PL=1
MOVL C00956 V=30.0 PL=1
MOVL C00957 V=30.0 PL=1
MOVL C00958 V=30.0 PL=1
MOVL C00959 V=30.0 PL=1
MOVL C00960 V=30.0 PL=1
MOVL C00961 V=30.0 PL=1
MOVL C00962 V=30.0 PL=1
MOVL C00963 V=30.0 PL=1
MOVL C00964 V=30.0 PL=1
MOVL C00965 V=30.0 PL=1
MOVL C00966 V=30.0 PL=1
MOVL C00967 V=30.0 PL=1
MOVL C00968 V=30.0 PL=1
MOVL C00969 V=30.0 PL=1
MOVL C00970 V=30.0 PL=1
MOVL C00971 V=30.0 PL=1
MOVL C00972 V=30.0 PL=1
MOVL C00973 V=30.0 PL=1
MOVL C00974 V=30.0 PL=1
MOVL C00975 V=30.0 PL=1
MOVL C00976 V=30.0 PL=1
MOVL C00977 V=30.0 PL=1
MOVL C00978 V=30.0 PL=1
MOVL C00979 V=30.0 PL=1
MOVL C00980 V=30.0 PL=1
MOVL C00981 V=30.0 PL=1
MOVL C00982 V=30.0 PL=1
MOVL C00983 V=30.0 PL=1
MOVL C00984 V=30.0 PL=1
MOVL C00985 V=30.0 PL=1
MOVL C00986 V=30.0 PL=1
MOVL C00987 V=30.0 PL=1
MOVL C00988 V=30.0 PL=1
MOVL C00989 V=30.0 PL=1
END
